	UF : 0, UT : 6,		CONFIG : 'N U T, 0, 0, 0',
	X =  19.695  mm,	Y =   -632.408  mm,	Z =   -236.035  mm,
	W =  90.000 deg,	P =   0.000 deg,	R =   90.000 deg
};
P[1150]{
   GP1:
	UF : 0, UT : 6,		CONFIG : 'N U T, 0, 0, 0',
	X =  20.066  mm,	Y =   -632.890  mm,	Z =   -236.261  mm,
	W =  90.000 deg,	P =   0.000 deg,	R =   90.000 deg
};
P[1151]{
   GP1:
	UF : 0, UT : 6,		CONFIG : 'N U T, 0, 0, 0',
	X =  21.473  mm,	Y =   -635.520  mm,	Z =   -235.987  mm,
	W =  90.000 deg,	P =   0.000 deg,	R =   90.000 deg
};
P[1152]{
   GP1:
	UF : 0, UT : 6,		CONFIG : 'N U T, 0, 0, 0',
	X =  22.170  mm,	Y =   -636.842  mm,	Z =   -235.830  mm,
	W =  90.000 deg,	P =   0.000 deg,	R =   90.000 deg
};
P[1153]{
   GP1:
	UF : 0, UT : 6,		CONFIG : 'N U T, 0, 0, 0',
	X =  22.857  mm,	Y =   -637.882  mm,	Z =   -236.036  mm,
	W =  90.000 deg,	P =   0.000 deg,	R =   90.000 deg
};
P[1154]{
   GP1:
	UF : 0, UT : 6,		CONFIG : 'N U T, 0, 0, 0',
	X =  25.259  mm,	Y =   -642.193  mm,	Z =   -235.826  mm,
	W =  90.000 deg,	P =   0.000 deg,	R =   90.000 deg
};
P[1155]{
   GP1:
	UF : 0, UT : 6,		CONFIG : 'N U T, 0, 0, 0',
	X =  26.183  mm,	Y =   -643.553  mm,	Z =   -236.163  mm,
	W =  90.000 deg,	P =   0.000 deg,	R =   90.000 deg
};
P[1156]{
   GP1:
	UF : 0, UT : 6,		CONFIG : 'N U T, 0, 0, 0',
	X =  26.417  mm,	Y =   -644.215  mm,	Z =   -235.804  mm,
	W =  90.000 deg,	P =   0.000 deg,	R =   90.000 deg
};
P[1157]{
   GP1:
	UF : 0, UT : 6,		CONFIG : 'N U T, 0, 0, 0',
	X =  27.412  mm,	Y =   -645.826  mm,	Z =   -235.959  mm,
	W =  90.000 deg,	P =   0.000 deg,	R =   90.000 deg
};
P[1158]{
   GP1:
	UF : 0, UT : 6,		CONFIG : 'N U T, 0, 0, 0',
	X =  28.982  mm,	Y =   -648.431  mm,	Z =   -236.122  mm,
	W =  90.000 deg,	P =   0.000 deg,	R =   90.000 deg
};
P[1159]{
   GP1:
	UF : 0, UT : 6,		CONFIG : 'N U T, 0, 0, 0',
	X =  29.599  mm,	Y =   -649.401  mm,	Z =   -236.259  mm,
	W =  90.000 deg,	P =   0.000 deg,	R =   90.000 deg
};
P[1160]{
   GP1:
	UF : 0, UT : 6,		CONFIG : 'N U T, 0, 0, 0',
	X =  30.088  mm,	Y =   -650.463  mm,	Z =   -235.958  mm,
	W =  90.000 deg,	P =   0.000 deg,	R =   90.000 deg
};
P[1161]{
   GP1:
	UF : 0, UT : 6,		CONFIG : 'N U T, 0, 0, 0',
	X =  30.788  mm,	Y =   -651.725  mm,	Z =   -235.889  mm,
	W =  90.000 deg,	P =   0.000 deg,	R =   90.000 deg
};
P[1162]{
   GP1:
	UF : 0, UT : 6,		CONFIG : 'N U T, 0, 0, 0',
	X =  31.326  mm,	Y =   -652.437  mm,	Z =   -236.196  mm,
	W =  90.000 deg,	P =   0.000 deg,	R =   90.000 deg
};
P[1163]{
   GP1:
	UF : 0, UT : 6,		CONFIG : 'N U T, 0, 0, 0',
	X =  33.837  mm,	Y =   -656.822  mm,	Z =   -236.144  mm,
	W =  90.000 deg,	P =   0.000 deg,	R =   90.000 deg
};
P[1164]{
   GP1:
	UF : 0, UT : 6,		CONFIG : 'N U T, 0, 0, 0',
	X =  34.171  mm,	Y =   -657.333  mm,	Z =   -236.240  mm,
	W =  90.000 deg,	P =   0.000 deg,	R =   90.000 deg
};
P[1165]{
   GP1:
	UF : 0, UT : 6,		CONFIG : 'N U T, 0, 0, 0',
	X =  35.312  mm,	Y =   -659.302  mm,	Z =   -236.251  mm,
	W =  90.000 deg,	P =   0.000 deg,	R =   90.000 deg
};
P[1166]{
   GP1:
	UF : 0, UT : 6,		CONFIG : 'N U T, 0, 0, 0',
	X =  36.261  mm,	Y =   -661.175  mm,	Z =   -235.927  mm,
	W =  90.000 deg,	P =   0.000 deg,	R =   90.000 deg
};
P[1167]{
   GP1:
	UF : 0, UT : 6,		CONFIG : 'N U T, 0, 0, 0',
	X =  36.673  mm,	Y =   -661.862  mm,	Z =   -235.965  mm,
	W =  90.000 deg,	P =   0.000 deg,	R =   90.000 deg
};
P[1168]{
   GP1:
	UF : 0, UT : 6,		CONFIG : 'N U T, 0, 0, 0',
	X =  37.452  mm,	Y =   -663.236  mm,	Z =   -235.932  mm,
	W =  90.000 deg,	P =   0.000 deg,	R =   90.000 deg
};
P[1169]{
   GP1:
	UF : 0, UT : 6,		CONFIG : 'N U T, 0, 0, 0',
	X =  38.851  mm,	Y =   -665.730  mm,	Z =   -235.831  mm,
	W =  90.000 deg,	P =   0.000 deg,	R =   90.000 deg
};
P[1170]{
   GP1:
	UF : 0, UT : 6,		CONFIG : 'N U T, 0, 0, 0',
	X =  39.817  mm,	Y =   -667.148  mm,	Z =   -236.188  mm,
	W =  90.000 deg,	P =   0.000 deg,	R =   90.000 deg
};
P[1171]{
   GP1:
	UF : 0, UT : 6,		CONFIG : 'N U T, 0, 0, 0',
	X =  41.225  mm,	Y =   -669.627  mm,	Z =   -236.131  mm,
	W =  90.000 deg,	P =   0.000 deg,	R =   90.000 deg
};
P[1172]{
   GP1:
	UF : 0, UT : 6,		CONFIG : 'N U T, 0, 0, 0',
	X =  41.505  mm,	Y =   -670.293  mm,	Z =   -235.877  mm,
	W =  90.000 deg,	P =   0.000 deg,	R =   90.000 deg
};
P[1173]{
   GP1:
	UF : 0, UT : 6,		CONFIG : 'N U T, 0, 0, 0',
	X =  42.466  mm,	Y =   -671.763  mm,	Z =   -236.150  mm,
	W =  90.000 deg,	P =   0.000 deg,	R =   90.000 deg
};
P[1174]{
   GP1:
	UF : 0, UT : 6,		CONFIG : 'N U T, 0, 0, 0',
	X =  44.206  mm,	Y =   -675.025  mm,	Z =   -235.802  mm,
	W =  90.000 deg,	P =   0.000 deg,	R =   90.000 deg
};
P[1175]{
   GP1:
	UF : 0, UT : 6,		CONFIG : 'N U T, 0, 0, 0',
	X =  45.308  mm,	Y =   -676.876  mm,	Z =   -235.884  mm,
	W =  90.000 deg,	P =   0.000 deg,	R =   90.000 deg
};
P[1176]{
   GP1:
	UF : 0, UT : 6,		CONFIG : 'N U T, 0, 0, 0',
	X =  48.322  mm,	Y =   -681.161  mm,	Z =   -236.219  mm,
	W =  90.000 deg,	P =   0.000 deg,	R =   90.000 deg
};
P[1177]{
   GP1:
	UF : 0, UT : 6,		CONFIG : 'N U T, 0, 0, 0',
	X =  48.985  mm,	Y =   -682.066  mm,	Z =   -235.767  mm,
	W =  90.000 deg,	P =   0.000 deg,	R =   90.000 deg
};
P[1178]{
   GP1:
	UF : 0, UT : 6,		CONFIG : 'N U T, 0, 0, 0',
	X =  50.468  mm,	Y =   -683.145  mm,	Z =   -236.020  mm,
	W =  90.000 deg,	P =   0.000 deg,	R =   90.000 deg
};
P[1179]{
   GP1:
	UF : 0, UT : 6,		CONFIG : 'N U T, 0, 0, 0',
	X =  52.789  mm,	Y =   -684.503  mm,	Z =   -235.854  mm,
	W =  90.000 deg,	P =   0.000 deg,	R =   90.000 deg
};
P[1180]{
   GP1:
	UF : 0, UT : 6,		CONFIG : 'N U T, 0, 0, 0',
	X =  57.085  mm,	Y =   -685.239  mm,	Z =   -236.177  mm,
	W =  90.000 deg,	P =   0.000 deg,	R =   90.000 deg
};
P[1181]{
   GP1:
	UF : 0, UT : 6,		CONFIG : 'N U T, 0, 0, 0',
	X =  59.311  mm,	Y =   -685.278  mm,	Z =   -235.865  mm,
	W =  90.000 deg,	P =   0.000 deg,	R =   90.000 deg
};
P[1182]{
   GP1:
	UF : 0, UT : 6,		CONFIG : 'N U T, 0, 0, 0',
	X =  60.413  mm,	Y =   -684.908  mm,	Z =   -236.185  mm,
	W =  90.000 deg,	P =   0.000 deg,	R =   90.000 deg
};
P[1183]{
   GP1:
	UF : 0, UT : 6,		CONFIG : 'N U T, 0, 0, 0',
	X =  61.691  mm,	Y =   -684.746  mm,	Z =   -235.808  mm,
	W =  90.000 deg,	P =   0.000 deg,	R =   90.000 deg
};
P[1184]{
   GP1:
	UF : 0, UT : 6,		CONFIG : 'N U T, 0, 0, 0',
	X =  62.508  mm,	Y =   -684.214  mm,	Z =   -236.201  mm,
	W =  90.000 deg,	P =   0.000 deg,	R =   90.000 deg
};
P[1185]{
   GP1:
	UF : 0, UT : 6,		CONFIG : 'N U T, 0, 0, 0',
	X =  63.457  mm,	Y =   -683.779  mm,	Z =   -236.224  mm,
	W =  90.000 deg,	P =   0.000 deg,	R =   90.000 deg
};
P[1186]{
   GP1:
	UF : 0, UT : 6,		CONFIG : 'N U T, 0, 0, 0',
	X =  64.865  mm,	Y =   -683.047  mm,	Z =   -236.231  mm,
	W =  90.000 deg,	P =   0.000 deg,	R =   90.000 deg
};
P[1187]{
   GP1:
	UF : 0, UT : 6,		CONFIG : 'N U T, 0, 0, 0',
	X =  66.260  mm,	Y =   -682.344  mm,	Z =   -235.984  mm,
	W =  90.000 deg,	P =   0.000 deg,	R =   90.000 deg
};
P[1188]{
   GP1:
	UF : 0, UT : 6,		CONFIG : 'N U T, 0, 0, 0',
	X =  68.438  mm,	Y =   -681.119  mm,	Z =   -235.906  mm,
	W =  90.000 deg,	P =   0.000 deg,	R =   90.000 deg
};
P[1189]{
   GP1:
	UF : 0, UT : 6,		CONFIG : 'N U T, 0, 0, 0',
	X =  71.774  mm,	Y =   -679.075  mm,	Z =   -236.192  mm,
	W =  90.000 deg,	P =   0.000 deg,	R =   90.000 deg
};
P[1190]{
   GP1:
	UF : 0, UT : 6,		CONFIG : 'N U T, 0, 0, 0',
	X =  72.829  mm,	Y =   -678.491  mm,	Z =   -236.131  mm,
	W =  90.000 deg,	P =   0.000 deg,	R =   90.000 deg
};
P[1191]{
   GP1:
	UF : 0, UT : 6,		CONFIG : 'N U T, 0, 0, 0',
	X =  75.444  mm,	Y =   -677.073  mm,	Z =   -235.905  mm,
	W =  90.000 deg,	P =   0.000 deg,	R =   90.000 deg
};
P[1192]{
   GP1:
	UF : 0, UT : 6,		CONFIG : 'N U T, 0, 0, 0',
	X =  76.617  mm,	Y =   -676.318  mm,	Z =   -236.096  mm,
	W =  90.000 deg,	P =   0.000 deg,	R =   90.000 deg
};
P[1193]{
   GP1:
	UF : 0, UT : 6,		CONFIG : 'N U T, 0, 0, 0',
	X =  82.666  mm,	Y =   -672.836  mm,	Z =   -236.069  mm,
	W =  90.000 deg,	P =   0.000 deg,	R =   90.000 deg
};
P[1194]{
   GP1:
	UF : 0, UT : 6,		CONFIG : 'N U T, 0, 0, 0',
	X =  83.579  mm,	Y =   -672.339  mm,	Z =   -235.997  mm,
	W =  90.000 deg,	P =   0.000 deg,	R =   90.000 deg
};
P[1195]{
   GP1:
	UF : 0, UT : 6,		CONFIG : 'N U T, 0, 0, 0',
	X =  84.352  mm,	Y =   -671.819  mm,	Z =   -236.176  mm,
	W =  90.000 deg,	P =   0.000 deg,	R =   90.000 deg
};
P[1196]{
   GP1:
	UF : 0, UT : 6,		CONFIG : 'N U T, 0, 0, 0',
	X =  86.806  mm,	Y =   -670.389  mm,	Z =   -236.207  mm,
	W =  90.000 deg,	P =   0.000 deg,	R =   90.000 deg
};
P[1197]{
   GP1:
	UF : 0, UT : 6,		CONFIG : 'N U T, 0, 0, 0',
	X =  87.702  mm,	Y =   -669.881  mm,	Z =   -236.187  mm,
	W =  90.000 deg,	P =   0.000 deg,	R =   90.000 deg
};
P[1198]{
   GP1:
	UF : 0, UT : 6,		CONFIG : 'N U T, 0, 0, 0',
	X =  91.684  mm,	Y =   -667.560  mm,	Z =   -236.236  mm,
	W =  90.000 deg,	P =   0.000 deg,	R =   90.000 deg
};
P[1199]{
   GP1:
	UF : 0, UT : 6,		CONFIG : 'N U T, 0, 0, 0',
	X =  92.871  mm,	Y =   -666.995  mm,	Z =   -235.945  mm,
	W =  90.000 deg,	P =   0.000 deg,	R =   90.000 deg
};
P[1200]{
   GP1:
	UF : 0, UT : 6,		CONFIG : 'N U T, 0, 0, 0',
	X =  93.918  mm,	Y =   -666.295  mm,	Z =   -236.177  mm,
	W =  90.000 deg,	P =   0.000 deg,	R =   90.000 deg
};
P[1201]{
   GP1:
	UF : 0, UT : 6,		CONFIG : 'N U T, 0, 0, 0',
	X =  96.550  mm,	Y =   -664.748  mm,	Z =   -236.242  mm,
	W =  90.000 deg,	P =   0.000 deg,	R =   90.000 deg
};
P[1202]{
   GP1:
	UF : 0, UT : 6,		CONFIG : 'N U T, 0, 0, 0',
	X =  98.885  mm,	Y =   -663.545  mm,	Z =   -235.890  mm,
	W =  90.000 deg,	P =   0.000 deg,	R =   90.000 deg
};
P[1203]{
   GP1:
	UF : 0, UT : 6,		CONFIG : 'N U T, 0, 0, 0',
	X =  101.949  mm,	Y =   -661.786  mm,	Z =   -235.866  mm,
	W =  90.000 deg,	P =   0.000 deg,	R =   90.000 deg
};
P[1204]{
   GP1:
	UF : 0, UT : 6,		CONFIG : 'N U T, 0, 0, 0',
	X =  105.049  mm,	Y =   -659.837  mm,	Z =   -236.252  mm,
	W =  90.000 deg,	P =   0.000 deg,	R =   90.000 deg
};
P[1205]{
   GP1:
	UF : 0, UT : 6,		CONFIG : 'N U T, 0, 0, 0',
	X =  107.967  mm,	Y =   -658.192  mm,	Z =   -236.155  mm,
	W =  90.000 deg,	P =   0.000 deg,	R =   90.000 deg
};
P[1206]{
   GP1:
	UF : 0, UT : 6,		CONFIG : 'N U T, 0, 0, 0',
	X =  109.064  mm,	Y =   -657.606  mm,	Z =   -236.039  mm,
	W =  90.000 deg,	P =   0.000 deg,	R =   90.000 deg
};
P[1207]{
   GP1:
	UF : 0, UT : 6,		CONFIG : 'N U T, 0, 0, 0',
	X =  110.455  mm,	Y =   -656.731  mm,	Z =   -236.216  mm,
	W =  90.000 deg,	P =   0.000 deg,	R =   90.000 deg
};
P[1208]{
   GP1:
	UF : 0, UT : 6,		CONFIG : 'N U T, 0, 0, 0',
	X =  113.229  mm,	Y =   -655.189  mm,	Z =   -236.069  mm,
	W =  90.000 deg,	P =   0.000 deg,	R =   90.000 deg
};
P[1209]{
   GP1:
	UF : 0, UT : 6,		CONFIG : 'N U T, 0, 0, 0',
	X =  115.613  mm,	Y =   -653.845  mm,	Z =   -235.990  mm,
	W =  90.000 deg,	P =   0.000 deg,	R =   90.000 deg
};
P[1210]{
   GP1:
	UF : 0, UT : 6,		CONFIG : 'N U T, 0, 0, 0',
	X =  120.896  mm,	Y =   -650.754  mm,	Z =   -236.090  mm,
	W =  90.000 deg,	P =   0.000 deg,	R =   90.000 deg
};
P[1211]{
   GP1:
	UF : 0, UT : 6,		CONFIG : 'N U T, 0, 0, 0',
	X =  122.286  mm,	Y =   -649.951  mm,	Z =   -236.092  mm,
	W =  90.000 deg,	P =   0.000 deg,	R =   90.000 deg
};
P[1212]{
   GP1:
	UF : 0, UT : 6,		CONFIG : 'N U T, 0, 0, 0',
	X =  128.537  mm,	Y =   -646.275  mm,	Z =   -236.252  mm,
	W =  90.000 deg,	P =   0.000 deg,	R =   90.000 deg
};
P[1213]{
   GP1:
	UF : 0, UT : 6,		CONFIG : 'N U T, 0, 0, 0',
	X =  129.609  mm,	Y =   -645.663  mm,	Z =   -236.237  mm,
	W =  90.000 deg,	P =   0.000 deg,	R =   90.000 deg
};
P[1214]{
   GP1:
	UF : 0, UT : 6,		CONFIG : 'N U T, 0, 0, 0',
	X =  130.636  mm,	Y =   -645.107  mm,	Z =   -236.148  mm,
	W =  90.000 deg,	P =   0.000 deg,	R =   90.000 deg
};
P[1215]{
   GP1:
	UF : 0, UT : 6,		CONFIG : 'N U T, 0, 0, 0',
	X =  131.238  mm,	Y =   -644.736  mm,	Z =   -236.204  mm,
	W =  90.000 deg,	P =   0.000 deg,	R =   90.000 deg
};
P[1216]{
   GP1:
	UF : 0, UT : 6,		CONFIG : 'N U T, 0, 0, 0',
	X =  135.205  mm,	Y =   -642.495  mm,	Z =   -236.084  mm,
	W =  90.000 deg,	P =   0.000 deg,	R =   90.000 deg
};
P[1217]{
   GP1:
	UF : 0, UT : 6,		CONFIG : 'N U T, 0, 0, 0',
	X =  138.112  mm,	Y =   -640.947  mm,	Z =   -235.765  mm,
	W =  90.000 deg,	P =   0.000 deg,	R =   90.000 deg
};
P[1218]{
   GP1:
	UF : 0, UT : 6,		CONFIG : 'N U T, 0, 0, 0',
	X =  139.022  mm,	Y =   -640.231  mm,	Z =   -236.231  mm,
	W =  90.000 deg,	P =   0.000 deg,	R =   90.000 deg
};
P[1219]{
   GP1:
	UF : 0, UT : 6,		CONFIG : 'N U T, 0, 0, 0',
	X =  140.803  mm,	Y =   -639.313  mm,	Z =   -235.959  mm,
	W =  90.000 deg,	P =   0.000 deg,	R =   90.000 deg
};
P[1220]{
   GP1:
	UF : 0, UT : 6,		CONFIG : 'N U T, 0, 0, 0',
	X =  141.464  mm,	Y =   -638.891  mm,	Z =   -236.060  mm,
	W =  90.000 deg,	P =   0.000 deg,	R =   90.000 deg
};
P[1221]{
   GP1:
	UF : 0, UT : 6,		CONFIG : 'N U T, 0, 0, 0',
	X =  144.134  mm,	Y =   -637.401  mm,	Z =   -235.935  mm,
	W =  90.000 deg,	P =   0.000 deg,	R =   90.000 deg
};
P[1222]{
   GP1:
	UF : 0, UT : 6,		CONFIG : 'N U T, 0, 0, 0',
	X =  145.036  mm,	Y =   -636.806  mm,	Z =   -236.112  mm,
	W =  90.000 deg,	P =   0.000 deg,	R =   90.000 deg
};
P[1223]{
   GP1:
	UF : 0, UT : 6,		CONFIG : 'N U T, 0, 0, 0',
	X =  145.813  mm,	Y =   -636.296  mm,	Z =   -236.263  mm,
	W =  90.000 deg,	P =   0.000 deg,	R =   90.000 deg
};
P[1224]{
   GP1:
	UF : 0, UT : 6,		CONFIG : 'N U T, 0, 0, 0',
	X =  147.022  mm,	Y =   -635.665  mm,	Z =   -236.101  mm,
	W =  90.000 deg,	P =   0.000 deg,	R =   90.000 deg
};
P[1225]{
   GP1:
	UF : 0, UT : 6,		CONFIG : 'N U T, 0, 0, 0',
	X =  148.140  mm,	Y =   -635.017  mm,	Z =   -236.107  mm,
	W =  90.000 deg,	P =   0.000 deg,	R =   90.000 deg
};
P[1226]{
   GP1:
	UF : 0, UT : 6,		CONFIG : 'N U T, 0, 0, 0',
	X =  149.297  mm,	Y =   -634.466  mm,	Z =   -235.820  mm,
	W =  90.000 deg,	P =   0.000 deg,	R =   90.000 deg
};
P[1227]{
   GP1:
	UF : 0, UT : 6,		CONFIG : 'N U T, 0, 0, 0',
	X =  152.287  mm,	Y =   -632.743  mm,	Z =   -235.814  mm,
	W =  90.000 deg,	P =   0.000 deg,	R =   90.000 deg
};
P[1228]{
   GP1:
	UF : 0, UT : 6,		CONFIG : 'N U T, 0, 0, 0',
	X =  153.491  mm,	Y =   -631.907  mm,	Z =   -236.155  mm,
	W =  90.000 deg,	P =   0.000 deg,	R =   90.000 deg
};
P[1229]{
   GP1:
	UF : 0, UT : 6,		CONFIG : 'N U T, 0, 0, 0',
	X =  154.682  mm,	Y =   -631.302  mm,	Z =   -235.956  mm,
	W =  90.000 deg,	P =   0.000 deg,	R =   90.000 deg
};
P[1230]{
   GP1:
	UF : 0, UT : 6,		CONFIG : 'N U T, 0, 0, 0',
	X =  155.626  mm,	Y =   -630.706  mm,	Z =   -236.079  mm,
	W =  90.000 deg,	P =   0.000 deg,	R =   90.000 deg
};
P[1231]{
   GP1:
	UF : 0, UT : 6,		CONFIG : 'N U T, 0, 0, 0',
	X =  157.770  mm,	Y =   -629.514  mm,	Z =   -235.969  mm,
	W =  90.000 deg,	P =   0.000 deg,	R =   90.000 deg
};
P[1232]{
   GP1:
	UF : 0, UT : 6,		CONFIG : 'N U T, 0, 0, 0',
	X =  160.528  mm,	Y =   -627.937  mm,	Z =   -235.928  mm,
	W =  90.000 deg,	P =   0.000 deg,	R =   90.000 deg
};
P[1233]{
   GP1:
	UF : 0, UT : 6,		CONFIG : 'N U T, 0, 0, 0',
	X =  161.238  mm,	Y =   -627.424  mm,	Z =   -236.177  mm,
	W =  90.000 deg,	P =   0.000 deg,	R =   90.000 deg
};
P[1234]{
   GP1:
	UF : 0, UT : 6,		CONFIG : 'N U T, 0, 0, 0',
	X =  162.012  mm,	Y =   -627.052  mm,	Z =   -235.999  mm,
	W =  90.000 deg,	P =   0.000 deg,	R =   90.000 deg
};
P[1235]{
   GP1:
	UF : 0, UT : 6,		CONFIG : 'N U T, 0, 0, 0',
	X =  166.933  mm,	Y =   -624.102  mm,	Z =   -236.262  mm,
	W =  90.000 deg,	P =   0.000 deg,	R =   90.000 deg
};
P[1236]{
   GP1:
	UF : 0, UT : 6,		CONFIG : 'N U T, 0, 0, 0',
	X =  167.569  mm,	Y =   -623.749  mm,	Z =   -236.228  mm,
	W =  90.000 deg,	P =   0.000 deg,	R =   90.000 deg
};
P[1237]{
   GP1:
	UF : 0, UT : 6,		CONFIG : 'N U T, 0, 0, 0',
	X =  170.488  mm,	Y =   -622.121  mm,	Z =   -236.089  mm,
	W =  90.000 deg,	P =   0.000 deg,	R =   90.000 deg
};
P[1238]{
   GP1:
	UF : 0, UT : 6,		CONFIG : 'N U T, 0, 0, 0',
	X =  171.115  mm,	Y =   -621.725  mm,	Z =   -236.171  mm,
	W =  90.000 deg,	P =   0.000 deg,	R =   90.000 deg
};
P[1239]{
   GP1:
	UF : 0, UT : 6,		CONFIG : 'N U T, 0, 0, 0',
	X =  171.685  mm,	Y =   -621.363  mm,	Z =   -236.249  mm,
	W =  90.000 deg,	P =   0.000 deg,	R =   90.000 deg
};
P[1240]{
   GP1:
	UF : 0, UT : 6,		CONFIG : 'N U T, 0, 0, 0',
	X =  176.974  mm,	Y =   -618.470  mm,	Z =   -235.859  mm,
	W =  90.000 deg,	P =   0.000 deg,	R =   90.000 deg
};
P[1241]{
   GP1:
	UF : 0, UT : 6,		CONFIG : 'N U T, 0, 0, 0',
	X =  178.817  mm,	Y =   -617.389  mm,	Z =   -235.902  mm,
	W =  90.000 deg,	P =   0.000 deg,	R =   90.000 deg
};
P[1242]{
   GP1:
	UF : 0, UT : 6,		CONFIG : 'N U T, 0, 0, 0',
	X =  182.698  mm,	Y =   -615.137  mm,	Z =   -235.927  mm,
	W =  90.000 deg,	P =   0.000 deg,	R =   90.000 deg
};
P[1243]{
   GP1:
	UF : 0, UT : 6,		CONFIG : 'N U T, 0, 0, 0',
	X =  187.118  mm,	Y =   -612.467  mm,	Z =   -236.214  mm,
	W =  90.000 deg,	P =   0.000 deg,	R =   90.000 deg
};
P[1244]{
   GP1:
	UF : 0, UT : 6,		CONFIG : 'N U T, 0, 0, 0',
	X =  190.558  mm,	Y =   -610.460  mm,	Z =   -236.263  mm,
	W =  90.000 deg,	P =   0.000 deg,	R =   90.000 deg
};
P[1245]{
   GP1:
	UF : 0, UT : 6,		CONFIG : 'N U T, 0, 0, 0',
	X =  194.089  mm,	Y =   -608.591  mm,	Z =   -235.851  mm,
	W =  90.000 deg,	P =   0.000 deg,	R =   90.000 deg
};
P[1246]{
   GP1:
	UF : 0, UT : 6,		CONFIG : 'N U T, 0, 0, 0',
	X =  195.296  mm,	Y =   -607.726  mm,	Z =   -236.259  mm,
	W =  90.000 deg,	P =   0.000 deg,	R =   90.000 deg
};
P[1247]{
   GP1:
	UF : 0, UT : 6,		CONFIG : 'N U T, 0, 0, 0',
	X =  197.817  mm,	Y =   -606.299  mm,	Z =   -236.192  mm,
	W =  90.000 deg,	P =   0.000 deg,	R =   90.000 deg
};
P[1248]{
   GP1:
	UF : 0, UT : 6,		CONFIG : 'N U T, 0, 0, 0',
	X =  201.527  mm,	Y =   -604.217  mm,	Z =   -236.045  mm,
	W =  90.000 deg,	P =   0.000 deg,	R =   90.000 deg
};
P[1249]{
   GP1:
	UF : 0, UT : 6,		CONFIG : 'N U T, 0, 0, 0',
	X =  203.422  mm,	Y =   -603.063  mm,	Z =   -236.190  mm,
	W =  90.000 deg,	P =   0.000 deg,	R =   90.000 deg
};
P[1250]{
   GP1:
	UF : 0, UT : 6,		CONFIG : 'N U T, 0, 0, 0',
	X =  205.460  mm,	Y =   -602.039  mm,	Z =   -235.818  mm,
	W =  90.000 deg,	P =   0.000 deg,	R =   90.000 deg
};
P[1251]{
   GP1:
	UF : 0, UT : 6,		CONFIG : 'N U T, 0, 0, 0',
	X =  207.396  mm,	Y =   -600.770  mm,	Z =   -236.186  mm,
	W =  90.000 deg,	P =   0.000 deg,	R =   90.000 deg
};
P[1252]{
   GP1:
	UF : 0, UT : 6,		CONFIG : 'N U T, 0, 0, 0',
	X =  208.921  mm,	Y =   -599.898  mm,	Z =   -236.166  mm,
	W =  90.000 deg,	P =   0.000 deg,	R =   90.000 deg
};
P[1253]{
   GP1:
	UF : 0, UT : 6,		CONFIG : 'N U T, 0, 0, 0',
	X =  214.058  mm,	Y =   -596.930  mm,	Z =   -236.170  mm,
	W =  90.000 deg,	P =   0.000 deg,	R =   90.000 deg
};
P[1254]{
   GP1:
	UF : 0, UT : 6,		CONFIG : 'N U T, 0, 0, 0',
	X =  215.411  mm,	Y =   -596.265  mm,	Z =   -235.888  mm,
	W =  90.000 deg,	P =   0.000 deg,	R =   90.000 deg
};
P[1255]{
   GP1:
	UF : 0, UT : 6,		CONFIG : 'N U T, 0, 0, 0',
	X =  216.083  mm,	Y =   -595.781  mm,	Z =   -236.121  mm,
	W =  90.000 deg,	P =   0.000 deg,	R =   90.000 deg
};
P[1256]{
   GP1:
	UF : 0, UT : 6,		CONFIG : 'N U T, 0, 0, 0',
	X =  217.510  mm,	Y =   -595.040  mm,	Z =   -235.921  mm,
	W =  90.000 deg,	P =   0.000 deg,	R =   90.000 deg
};
P[1257]{
   GP1:
	UF : 0, UT : 6,		CONFIG : 'N U T, 0, 0, 0',
	X =  218.922  mm,	Y =   -594.257  mm,	Z =   -235.842  mm,
	W =  90.000 deg,	P =   0.000 deg,	R =   90.000 deg
};
P[1258]{
   GP1:
	UF : 0, UT : 6,		CONFIG : 'N U T, 0, 0, 0',
	X =  220.028  mm,	Y =   -593.525  mm,	Z =   -236.068  mm,
	W =  90.000 deg,	P =   0.000 deg,	R =   90.000 deg
};
P[1259]{
   GP1:
	UF : 0, UT : 6,		CONFIG : 'N U T, 0, 0, 0',
	X =  220.868  mm,	Y =   -592.976  mm,	Z =   -236.224  mm,
	W =  90.000 deg,	P =   0.000 deg,	R =   90.000 deg
};
P[1260]{
   GP1:
	UF : 0, UT : 6,		CONFIG : 'N U T, 0, 0, 0',
	X =  221.717  mm,	Y =   -592.602  mm,	Z =   -235.941  mm,
	W =  90.000 deg,	P =   0.000 deg,	R =   90.000 deg
};
P[1261]{
   GP1:
	UF : 0, UT : 6,		CONFIG : 'N U T, 0, 0, 0',
	X =  227.339  mm,	Y =   -589.409  mm,	Z =   -235.814  mm,
	W =  90.000 deg,	P =   0.000 deg,	R =   90.000 deg
};
P[1262]{
   GP1:
	UF : 0, UT : 6,		CONFIG : 'N U T, 0, 0, 0',
	X =  227.893  mm,	Y =   -588.916  mm,	Z =   -236.232  mm,
	W =  90.000 deg,	P =   0.000 deg,	R =   90.000 deg
};
P[1263]{
   GP1:
	UF : 0, UT : 6,		CONFIG : 'N U T, 0, 0, 0',
	X =  229.324  mm,	Y =   -588.095  mm,	Z =   -236.219  mm,
	W =  90.000 deg,	P =   0.000 deg,	R =   90.000 deg
};
P[1264]{
   GP1:
	UF : 0, UT : 6,		CONFIG : 'N U T, 0, 0, 0',
	X =  230.255  mm,	Y =   -587.636  mm,	Z =   -236.030  mm,
	W =  90.000 deg,	P =   0.000 deg,	R =   90.000 deg
};
P[1265]{
   GP1:
	UF : 0, UT : 6,		CONFIG : 'N U T, 0, 0, 0',
	X =  231.063  mm,	Y =   -587.085  mm,	Z =   -236.234  mm,
	W =  90.000 deg,	P =   0.000 deg,	R =   90.000 deg
};
P[1266]{
   GP1:
	UF : 0, UT : 6,		CONFIG : 'N U T, 0, 0, 0',
	X =  232.274  mm,	Y =   -586.571  mm,	Z =   -235.786  mm,
	W =  90.000 deg,	P =   0.000 deg,	R =   90.000 deg
};
P[1267]{
   GP1:
	UF : 0, UT : 6,		CONFIG : 'N U T, 0, 0, 0',
	X =  234.541  mm,	Y =   -585.154  mm,	Z =   -236.047  mm,
	W =  90.000 deg,	P =   0.000 deg,	R =   90.000 deg
};
P[1268]{
   GP1:
	UF : 0, UT : 6,		CONFIG : 'N U T, 0, 0, 0',
	X =  235.154  mm,	Y =   -584.834  mm,	Z =   -235.966  mm,
	W =  90.000 deg,	P =   0.000 deg,	R =   90.000 deg
};
P[1269]{
   GP1:
	UF : 0, UT : 6,		CONFIG : 'N U T, 0, 0, 0',
	X =  238.918  mm,	Y =   -582.572  mm,	Z =   -236.180  mm,
	W =  90.000 deg,	P =   0.000 deg,	R =   90.000 deg
};
P[1270]{
   GP1:
	UF : 0, UT : 6,		CONFIG : 'N U T, 0, 0, 0',
	X =  240.565  mm,	Y =   -581.599  mm,	Z =   -236.235  mm,
	W =  90.000 deg,	P =   0.000 deg,	R =   90.000 deg
};
P[1271]{
   GP1:
	UF : 0, UT : 6,		CONFIG : 'N U T, 0, 0, 0',
	X =  243.237  mm,	Y =   -580.142  mm,	Z =   -236.025  mm,
	W =  90.000 deg,	P =   0.000 deg,	R =   90.000 deg
};
P[1272]{
   GP1:
	UF : 0, UT : 6,		CONFIG : 'N U T, 0, 0, 0',
	X =  243.899  mm,	Y =   -579.691  mm,	Z =   -236.193  mm,
	W =  90.000 deg,	P =   0.000 deg,	R =   90.000 deg
};
P[1273]{
   GP1:
	UF : 0, UT : 6,		CONFIG : 'N U T, 0, 0, 0',
	X =  246.134  mm,	Y =   -578.564  mm,	Z =   -235.796  mm,
	W =  90.000 deg,	P =   0.000 deg,	R =   90.000 deg
};
P[1274]{
   GP1:
	UF : 0, UT : 6,		CONFIG : 'N U T, 0, 0, 0',
	X =  246.789  mm,	Y =   -578.068  mm,	Z =   -236.081  mm,
	W =  90.000 deg,	P =   0.000 deg,	R =   90.000 deg
};
P[1275]{
   GP1:
	UF : 0, UT : 6,		CONFIG : 'N U T, 0, 0, 0',
	X =  248.147  mm,	Y =   -577.360  mm,	Z =   -235.895  mm,
	W =  90.000 deg,	P =   0.000 deg,	R =   90.000 deg
};
P[1276]{
   GP1:
	UF : 0, UT : 6,		CONFIG : 'N U T, 0, 0, 0',
	X =  250.469  mm,	Y =   -575.911  mm,	Z =   -236.160  mm,
	W =  90.000 deg,	P =   0.000 deg,	R =   90.000 deg
};
P[1277]{
   GP1:
	UF : 0, UT : 6,		CONFIG : 'N U T, 0, 0, 0',
	X =  250.972  mm,	Y =   -575.776  mm,	Z =   -235.783  mm,
	W =  90.000 deg,	P =   0.000 deg,	R =   90.000 deg
};
P[1278]{
   GP1:
	UF : 0, UT : 6,		CONFIG : 'N U T, 0, 0, 0',
	X =  251.820  mm,	Y =   -575.114  mm,	Z =   -236.201  mm,
	W =  90.000 deg,	P =   0.000 deg,	R =   90.000 deg
};
P[1279]{
   GP1:
	UF : 0, UT : 6,		CONFIG : 'N U T, 0, 0, 0',
	X =  253.992  mm,	Y =   -573.920  mm,	Z =   -236.056  mm,
	W =  90.000 deg,	P =   0.000 deg,	R =   90.000 deg
};
P[1280]{
   GP1:
	UF : 0, UT : 6,		CONFIG : 'N U T, 0, 0, 0',
	X =  255.262  mm,	Y =   -573.131  mm,	Z =   -236.189  mm,
	W =  90.000 deg,	P =   0.000 deg,	R =   90.000 deg
};
P[1281]{
   GP1:
	UF : 0, UT : 6,		CONFIG : 'N U T, 0, 0, 0',
	X =  257.360  mm,	Y =   -571.996  mm,	Z =   -236.003  mm,
	W =  90.000 deg,	P =   0.000 deg,	R =   90.000 deg
};
P[1282]{
   GP1:
	UF : 0, UT : 6,		CONFIG : 'N U T, 0, 0, 0',
	X =  258.170  mm,	Y =   -571.487  mm,	Z =   -236.104  mm,
	W =  90.000 deg,	P =   0.000 deg,	R =   90.000 deg
};
P[1283]{
   GP1:
	UF : 0, UT : 6,		CONFIG : 'N U T, 0, 0, 0',
	X =  258.767  mm,	Y =   -571.157  mm,	Z =   -236.070  mm,
	W =  90.000 deg,	P =   0.000 deg,	R =   90.000 deg
};
P[1284]{
   GP1:
	UF : 0, UT : 6,		CONFIG : 'N U T, 0, 0, 0',
	X =  260.090  mm,	Y =   -570.509  mm,	Z =   -235.789  mm,
	W =  90.000 deg,	P =   0.000 deg,	R =   90.000 deg
};
P[1285]{
   GP1:
	UF : 0, UT : 6,		CONFIG : 'N U T, 0, 0, 0',
	X =  261.709  mm,	Y =   -569.511  mm,	Z =   -235.943  mm,
	W =  90.000 deg,	P =   0.000 deg,	R =   90.000 deg
};
P[1286]{
   GP1:
	UF : 0, UT : 6,		CONFIG : 'N U T, 0, 0, 0',
	X =  264.842  mm,	Y =   -567.577  mm,	Z =   -236.245  mm,
	W =  90.000 deg,	P =   0.000 deg,	R =   90.000 deg
};
P[1287]{
   GP1:
	UF : 0, UT : 6,		CONFIG : 'N U T, 0, 0, 0',
	X =  266.479  mm,	Y =   -566.667  mm,	Z =   -236.161  mm,
	W =  90.000 deg,	P =   0.000 deg,	R =   90.000 deg
};
P[1288]{
   GP1:
	UF : 0, UT : 6,		CONFIG : 'N U T, 0, 0, 0',
	X =  267.664  mm,	Y =   -565.952  mm,	Z =   -236.234  mm,
	W =  90.000 deg,	P =   0.000 deg,	R =   90.000 deg
};
P[1289]{
   GP1:
	UF : 0, UT : 6,		CONFIG : 'N U T, 0, 0, 0',
	X =  276.056  mm,	Y =   -561.178  mm,	Z =   -236.061  mm,
	W =  90.000 deg,	P =   0.000 deg,	R =   90.000 deg
};
P[1290]{
   GP1:
	UF : 0, UT : 6,		CONFIG : 'N U T, 0, 0, 0',
	X =  277.168  mm,	Y =   -560.537  mm,	Z =   -236.057  mm,
	W =  90.000 deg,	P =   0.000 deg,	R =   90.000 deg
};
P[1291]{
   GP1:
	UF : 0, UT : 6,		CONFIG : 'N U T, 0, 0, 0',
	X =  283.306  mm,	Y =   -556.934  mm,	Z =   -236.202  mm,
	W =  90.000 deg,	P =   0.000 deg,	R =   90.000 deg
};
P[1292]{
   GP1:
	UF : 0, UT : 6,		CONFIG : 'N U T, 0, 0, 0',
	X =  283.968  mm,	Y =   -556.545  mm,	Z =   -236.217  mm,
	W =  90.000 deg,	P =   0.000 deg,	R =   90.000 deg
};
P[1293]{
   GP1:
	UF : 0, UT : 6,		CONFIG : 'N U T, 0, 0, 0',
	X =  285.871  mm,	Y =   -555.459  mm,	Z =   -236.187  mm,
	W =  90.000 deg,	P =   0.000 deg,	R =   90.000 deg
};
P[1294]{
   GP1:
	UF : 0, UT : 6,		CONFIG : 'N U T, 0, 0, 0',
	X =  287.181  mm,	Y =   -554.798  mm,	Z =   -235.956  mm,
	W =  90.000 deg,	P =   0.000 deg,	R =   90.000 deg
};
P[1295]{
   GP1:
	UF : 0, UT : 6,		CONFIG : 'N U T, 0, 0, 0',
	X =  288.139  mm,	Y =   -554.117  mm,	Z =   -236.265  mm,
	W =  90.000 deg,	P =   0.000 deg,	R =   90.000 deg
};
P[1296]{
   GP1:
	UF : 0, UT : 6,		CONFIG : 'N U T, 0, 0, 0',
	X =  289.724  mm,	Y =   -553.246  mm,	Z =   -236.158  mm,
	W =  90.000 deg,	P =   0.000 deg,	R =   90.000 deg
};
P[1297]{
   GP1:
	UF : 0, UT : 6,		CONFIG : 'N U T, 0, 0, 0',
	X =  291.588  mm,	Y =   -552.148  mm,	Z =   -236.211  mm,
	W =  90.000 deg,	P =   0.000 deg,	R =   90.000 deg
};
P[1298]{
   GP1:
	UF : 0, UT : 6,		CONFIG : 'N U T, 0, 0, 0',
	X =  295.641  mm,	Y =   -549.911  mm,	Z =   -235.963  mm,
	W =  90.000 deg,	P =   0.000 deg,	R =   90.000 deg
};
P[1299]{
   GP1:
	UF : 0, UT : 6,		CONFIG : 'N U T, 0, 0, 0',
	X =  296.764  mm,	Y =   -549.341  mm,	Z =   -235.771  mm,
	W =  90.000 deg,	P =   0.000 deg,	R =   90.000 deg
};
P[1300]{
   GP1:
	UF : 0, UT : 6,		CONFIG : 'N U T, 0, 0, 0',
	X =  297.702  mm,	Y =   -548.664  mm,	Z =   -236.100  mm,
	W =  90.000 deg,	P =   0.000 deg,	R =   90.000 deg
};
P[1301]{
   GP1:
	UF : 0, UT : 6,		CONFIG : 'N U T, 0, 0, 0',
	X =  299.074  mm,	Y =   -547.841  mm,	Z =   -236.174  mm,
	W =  90.000 deg,	P =   0.000 deg,	R =   90.000 deg
};
P[1302]{
   GP1:
	UF : 0, UT : 6,		CONFIG : 'N U T, 0, 0, 0',
	X =  302.115  mm,	Y =   -546.189  mm,	Z =   -235.922  mm,
	W =  90.000 deg,	P =   0.000 deg,	R =   90.000 deg
};
P[1303]{
   GP1:
	UF : 0, UT : 6,		CONFIG : 'N U T, 0, 0, 0',
	X =  304.281  mm,	Y =   -544.967  mm,	Z =   -235.853  mm,
	W =  90.000 deg,	P =   0.000 deg,	R =   90.000 deg
};
P[1304]{
   GP1:
	UF : 0, UT : 6,		CONFIG : 'N U T, 0, 0, 0',
	X =  305.391  mm,	Y =   -544.285  mm,	Z =   -235.952  mm,
	W =  90.000 deg,	P =   0.000 deg,	R =   90.000 deg
};
P[1305]{
   GP1:
	UF : 0, UT : 6,		CONFIG : 'N U T, 0, 0, 0',
	X =  307.431  mm,	Y =   -543.087  mm,	Z =   -236.003  mm,
	W =  90.000 deg,	P =   0.000 deg,	R =   90.000 deg
};
P[1306]{
   GP1:
	UF : 0, UT : 6,		CONFIG : 'N U T, 0, 0, 0',
	X =  311.087  mm,	Y =   -540.904  mm,	Z =   -236.176  mm,
	W =  90.000 deg,	P =   0.000 deg,	R =   90.000 deg
};
P[1307]{
   GP1:
	UF : 0, UT : 6,		CONFIG : 'N U T, 0, 0, 0',
	X =  313.813  mm,	Y =   -539.340  mm,	Z =   -236.153  mm,
	W =  90.000 deg,	P =   0.000 deg,	R =   90.000 deg
};
P[1308]{
   GP1:
	UF : 0, UT : 6,		CONFIG : 'N U T, 0, 0, 0',
	X =  316.236  mm,	Y =   -537.898  mm,	Z =   -236.255  mm,
	W =  90.000 deg,	P =   0.000 deg,	R =   90.000 deg
};
P[1309]{
   GP1:
	UF : 0, UT : 6,		CONFIG : 'N U T, 0, 0, 0',
	X =  317.798  mm,	Y =   -536.997  mm,	Z =   -236.256  mm,
	W =  90.000 deg,	P =   0.000 deg,	R =   90.000 deg
};
P[1310]{
   GP1:
	UF : 0, UT : 6,		CONFIG : 'N U T, 0, 0, 0',
	X =  318.889  mm,	Y =   -536.446  mm,	Z =   -236.063  mm,
	W =  90.000 deg,	P =   0.000 deg,	R =   90.000 deg
};
P[1311]{
   GP1:
	UF : 0, UT : 6,		CONFIG : 'N U T, 0, 0, 0',
	X =  319.712  mm,	Y =   -535.896  mm,	Z =   -236.245  mm,
	W =  90.000 deg,	P =   0.000 deg,	R =   90.000 deg
};
P[1312]{
   GP1:
	UF : 0, UT : 6,		CONFIG : 'N U T, 0, 0, 0',
	X =  321.761  mm,	Y =   -534.847  mm,	Z =   -235.919  mm,
	W =  90.000 deg,	P =   0.000 deg,	R =   90.000 deg
};
P[1313]{
   GP1:
	UF : 0, UT : 6,		CONFIG : 'N U T, 0, 0, 0',
	X =  323.593  mm,	Y =   -533.676  mm,	Z =   -236.192  mm,
	W =  90.000 deg,	P =   0.000 deg,	R =   90.000 deg
};
P[1314]{
   GP1:
	UF : 0, UT : 6,		CONFIG : 'N U T, 0, 0, 0',
	X =  328.811  mm,	Y =   -530.729  mm,	Z =   -236.034  mm,
	W =  90.000 deg,	P =   0.000 deg,	R =   90.000 deg
};
P[1315]{
   GP1:
	UF : 0, UT : 6,		CONFIG : 'N U T, 0, 0, 0',
	X =  331.545  mm,	Y =   -529.062  mm,	Z =   -236.246  mm,
	W =  90.000 deg,	P =   0.000 deg,	R =   90.000 deg
};
P[1316]{
   GP1:
	UF : 0, UT : 6,		CONFIG : 'N U T, 0, 0, 0',
	X =  332.941  mm,	Y =   -528.255  mm,	Z =   -236.250  mm,
	W =  90.000 deg,	P =   0.000 deg,	R =   90.000 deg
};
P[1317]{
   GP1:
	UF : 0, UT : 6,		CONFIG : 'N U T, 0, 0, 0',
	X =  336.586  mm,	Y =   -526.149  mm,	Z =   -236.254  mm,
	W =  90.000 deg,	P =   0.000 deg,	R =   90.000 deg
};
P[1318]{
   GP1:
	UF : 0, UT : 6,		CONFIG : 'N U T, 0, 0, 0',
	X =  339.977  mm,	Y =   -524.251  mm,	Z =   -236.109  mm,
	W =  90.000 deg,	P =   0.000 deg,	R =   90.000 deg
};
P[1319]{
   GP1:
	UF : 0, UT : 6,		CONFIG : 'N U T, 0, 0, 0',
	X =  341.795  mm,	Y =   -523.168  mm,	Z =   -236.189  mm,
	W =  90.000 deg,	P =   0.000 deg,	R =   90.000 deg
};
P[1320]{
   GP1:
	UF : 0, UT : 6,		CONFIG : 'N U T, 0, 0, 0',
	X =  342.831  mm,	Y =   -522.677  mm,	Z =   -235.930  mm,
	W =  90.000 deg,	P =   0.000 deg,	R =   90.000 deg
};
P[1321]{
   GP1:
	UF : 0, UT : 6,		CONFIG : 'N U T, 0, 0, 0',
	X =  343.741  mm,	Y =   -522.061  mm,	Z =   -236.148  mm,
	W =  90.000 deg,	P =   0.000 deg,	R =   90.000 deg
};
P[1322]{
   GP1:
	UF : 0, UT : 6,		CONFIG : 'N U T, 0, 0, 0',
	X =  347.154  mm,	Y =   -520.085  mm,	Z =   -236.164  mm,
	W =  90.000 deg,	P =   0.000 deg,	R =   90.000 deg
};
P[1323]{
   GP1:
	UF : 0, UT : 6,		CONFIG : 'N U T, 0, 0, 0',
	X =  349.167  mm,	Y =   -518.898  mm,	Z =   -236.221  mm,
	W =  90.000 deg,	P =   0.000 deg,	R =   90.000 deg
};
P[1324]{
   GP1:
	UF : 0, UT : 6,		CONFIG : 'N U T, 0, 0, 0',
	X =  352.757  mm,	Y =   -516.832  mm,	Z =   -236.203  mm,
	W =  90.000 deg,	P =   0.000 deg,	R =   90.000 deg
};
P[1325]{
   GP1:
	UF : 0, UT : 6,		CONFIG : 'N U T, 0, 0, 0',
	X =  356.030  mm,	Y =   -514.964  mm,	Z =   -236.152  mm,
	W =  90.000 deg,	P =   0.000 deg,	R =   90.000 deg
};
P[1326]{
   GP1:
	UF : 0, UT : 6,		CONFIG : 'N U T, 0, 0, 0',
	X =  357.181  mm,	Y =   -514.334  mm,	Z =   -236.069  mm,
	W =  90.000 deg,	P =   0.000 deg,	R =   90.000 deg
};
P[1327]{
   GP1:
	UF : 0, UT : 6,		CONFIG : 'N U T, 0, 0, 0',
	X =  358.019  mm,	Y =   -513.841  mm,	Z =   -236.091  mm,
	W =  90.000 deg,	P =   0.000 deg,	R =   90.000 deg
};
P[1328]{
   GP1:
	UF : 0, UT : 6,		CONFIG : 'N U T, 0, 0, 0',
	X =  358.836  mm,	Y =   -513.376  mm,	Z =   -236.075  mm,
	W =  90.000 deg,	P =   0.000 deg,	R =   90.000 deg
};
P[1329]{
   GP1:
	UF : 0, UT : 6,		CONFIG : 'N U T, 0, 0, 0',
	X =  359.384  mm,	Y =   -513.028  mm,	Z =   -236.152  mm,
	W =  90.000 deg,	P =   0.000 deg,	R =   90.000 deg
};
P[1330]{
   GP1:
	UF : 0, UT : 6,		CONFIG : 'N U T, 0, 0, 0',
	X =  360.335  mm,	Y =   -512.619  mm,	Z =   -235.811  mm,
	W =  90.000 deg,	P =   0.000 deg,	R =   90.000 deg
};
P[1331]{
   GP1:
	UF : 0, UT : 6,		CONFIG : 'N U T, 0, 0, 0',
	X =  362.804  mm,	Y =   -511.202  mm,	Z =   -235.789  mm,
	W =  90.000 deg,	P =   0.000 deg,	R =   90.000 deg
};
P[1332]{
   GP1:
	UF : 0, UT : 6,		CONFIG : 'N U T, 0, 0, 0',
	X =  364.805  mm,	Y =   -510.034  mm,	Z =   -235.820  mm,
	W =  90.000 deg,	P =   0.000 deg,	R =   90.000 deg
};
P[1333]{
   GP1:
	UF : 0, UT : 6,		CONFIG : 'N U T, 0, 0, 0',
	X =  365.931  mm,	Y =   -509.220  mm,	Z =   -236.218  mm,
	W =  90.000 deg,	P =   0.000 deg,	R =   90.000 deg
};
P[1334]{
   GP1:
	UF : 0, UT : 6,		CONFIG : 'N U T, 0, 0, 0',
	X =  366.787  mm,	Y =   -508.732  mm,	Z =   -236.203  mm,
	W =  90.000 deg,	P =   0.000 deg,	R =   90.000 deg
};
P[1335]{
   GP1:
	UF : 0, UT : 6,		CONFIG : 'N U T, 0, 0, 0',
	X =  369.185  mm,	Y =   -507.416  mm,	Z =   -236.037  mm,
	W =  90.000 deg,	P =   0.000 deg,	R =   90.000 deg
};
P[1336]{
   GP1:
	UF : 0, UT : 6,		CONFIG : 'N U T, 0, 0, 0',
	X =  370.161  mm,	Y =   -506.771  mm,	Z =   -236.235  mm,
	W =  90.000 deg,	P =   0.000 deg,	R =   90.000 deg
};
P[1337]{
   GP1:
	UF : 0, UT : 6,		CONFIG : 'N U T, 0, 0, 0',
	X =  370.741  mm,	Y =   -506.467  mm,	Z =   -236.161  mm,
	W =  90.000 deg,	P =   0.000 deg,	R =   90.000 deg
};
P[1338]{
   GP1:
	UF : 0, UT : 6,		CONFIG : 'N U T, 0, 0, 0',
	X =  373.216  mm,	Y =   -505.136  mm,	Z =   -235.923  mm,
	W =  90.000 deg,	P =   0.000 deg,	R =   90.000 deg
};
P[1339]{
   GP1:
	UF : 0, UT : 6,		CONFIG : 'N U T, 0, 0, 0',
	X =  373.769  mm,	Y =   -504.798  mm,	Z =   -235.968  mm,
	W =  90.000 deg,	P =   0.000 deg,	R =   90.000 deg
};
P[1340]{
   GP1:
	UF : 0, UT : 6,		CONFIG : 'N U T, 0, 0, 0',
	X =  375.268  mm,	Y =   -503.936  mm,	Z =   -235.961  mm,
	W =  90.000 deg,	P =   0.000 deg,	R =   90.000 deg
};
P[1341]{
   GP1:
	UF : 0, UT : 6,		CONFIG : 'N U T, 0, 0, 0',
	X =  376.365  mm,	Y =   -503.208  mm,	Z =   -236.189  mm,
	W =  90.000 deg,	P =   0.000 deg,	R =   90.000 deg
};
P[1342]{
   GP1:
	UF : 0, UT : 6,		CONFIG : 'N U T, 0, 0, 0',
	X =  377.812  mm,	Y =   -502.476  mm,	Z =   -235.937  mm,
	W =  90.000 deg,	P =   0.000 deg,	R =   90.000 deg
};
P[1343]{
   GP1:
	UF : 0, UT : 6,		CONFIG : 'N U T, 0, 0, 0',
	X =  378.644  mm,	Y =   -501.909  mm,	Z =   -236.149  mm,
	W =  90.000 deg,	P =   0.000 deg,	R =   90.000 deg
};
P[1344]{
   GP1:
	UF : 0, UT : 6,		CONFIG : 'N U T, 0, 0, 0',
	X =  382.006  mm,	Y =   -500.007  mm,	Z =   -236.051  mm,
	W =  90.000 deg,	P =   0.000 deg,	R =   90.000 deg
};
P[1345]{
   GP1:
	UF : 0, UT : 6,		CONFIG : 'N U T, 0, 0, 0',
	X =  384.094  mm,	Y =   -498.775  mm,	Z =   -236.118  mm,
	W =  90.000 deg,	P =   0.000 deg,	R =   90.000 deg
};
P[1346]{
   GP1:
	UF : 0, UT : 6,		CONFIG : 'N U T, 0, 0, 0',
	X =  385.040  mm,	Y =   -498.289  mm,	Z =   -235.969  mm,
	W =  90.000 deg,	P =   0.000 deg,	R =   90.000 deg
};
P[1347]{
   GP1:
	UF : 0, UT : 6,		CONFIG : 'N U T, 0, 0, 0',
	X =  387.969  mm,	Y =   -496.484  mm,	Z =   -236.245  mm,
	W =  90.000 deg,	P =   0.000 deg,	R =   90.000 deg
};
P[1348]{
   GP1:
	UF : 0, UT : 6,		CONFIG : 'N U T, 0, 0, 0',
	X =  388.653  mm,	Y =   -496.188  mm,	Z =   -236.005  mm,
	W =  90.000 deg,	P =   0.000 deg,	R =   90.000 deg
};
P[1349]{
   GP1:
	UF : 0, UT : 6,		CONFIG : 'N U T, 0, 0, 0',
	X =  389.771  mm,	Y =   -495.530  mm,	Z =   -236.036  mm,
	W =  90.000 deg,	P =   0.000 deg,	R =   90.000 deg
};
P[1350]{
   GP1:
	UF : 0, UT : 6,		CONFIG : 'N U T, 0, 0, 0',
	X =  391.734  mm,	Y =   -494.390  mm,	Z =   -236.054  mm,
	W =  90.000 deg,	P =   0.000 deg,	R =   90.000 deg
};
P[1351]{
   GP1:
	UF : 0, UT : 6,		CONFIG : 'N U T, 0, 0, 0',
	X =  393.563  mm,	Y =   -493.410  mm,	Z =   -235.867  mm,
	W =  90.000 deg,	P =   0.000 deg,	R =   90.000 deg
};
P[1352]{
   GP1:
	UF : 0, UT : 6,		CONFIG : 'N U T, 0, 0, 0',
	X =  395.191  mm,	Y =   -492.371  mm,	Z =   -236.108  mm,
	W =  90.000 deg,	P =   0.000 deg,	R =   90.000 deg
};
P[1353]{
   GP1:
	UF : 0, UT : 6,		CONFIG : 'N U T, 0, 0, 0',
	X =  395.783  mm,	Y =   -492.069  mm,	Z =   -236.013  mm,
	W =  90.000 deg,	P =   0.000 deg,	R =   90.000 deg
};
P[1354]{
   GP1:
	UF : 0, UT : 6,		CONFIG : 'N U T, 0, 0, 0',
	X =  396.375  mm,	Y =   -491.818  mm,	Z =   -235.791  mm,
	W =  90.000 deg,	P =   0.000 deg,	R =   90.000 deg
};
P[1355]{
   GP1:
	UF : 0, UT : 6,		CONFIG : 'N U T, 0, 0, 0',
	X =  397.057  mm,	Y =   -491.299  mm,	Z =   -236.097  mm,
	W =  90.000 deg,	P =   0.000 deg,	R =   90.000 deg
};
P[1356]{
   GP1:
	UF : 0, UT : 6,		CONFIG : 'N U T, 0, 0, 0',
	X =  398.898  mm,	Y =   -490.265  mm,	Z =   -236.024  mm,
	W =  90.000 deg,	P =   0.000 deg,	R =   90.000 deg
};
P[1357]{
   GP1:
	UF : 0, UT : 6,		CONFIG : 'N U T, 0, 0, 0',
	X =  399.925  mm,	Y =   -489.674  mm,	Z =   -236.019  mm,
	W =  90.000 deg,	P =   0.000 deg,	R =   90.000 deg
};
P[1358]{
   GP1:
	UF : 0, UT : 6,		CONFIG : 'N U T, 0, 0, 0',
	X =  401.212  mm,	Y =   -488.883  mm,	Z =   -236.137  mm,
	W =  90.000 deg,	P =   0.000 deg,	R =   90.000 deg
};
P[1359]{
   GP1:
	UF : 0, UT : 6,		CONFIG : 'N U T, 0, 0, 0',
	X =  403.329  mm,	Y =   -487.751  mm,	Z =   -235.916  mm,
	W =  90.000 deg,	P =   0.000 deg,	R =   90.000 deg
};
P[1360]{
   GP1:
	UF : 0, UT : 6,		CONFIG : 'N U T, 0, 0, 0',
	X =  403.952  mm,	Y =   -487.290  mm,	Z =   -236.163  mm,
	W =  90.000 deg,	P =   0.000 deg,	R =   90.000 deg
};
P[1361]{
   GP1:
	UF : 0, UT : 6,		CONFIG : 'N U T, 0, 0, 0',
	X =  404.904  mm,	Y =   -486.710  mm,	Z =   -236.237  mm,
	W =  90.000 deg,	P =   0.000 deg,	R =   90.000 deg
};
P[1362]{
   GP1:
	UF : 0, UT : 6,		CONFIG : 'N U T, 0, 0, 0',
	X =  406.898  mm,	Y =   -485.653  mm,	Z =   -236.006  mm,
	W =  90.000 deg,	P =   0.000 deg,	R =   90.000 deg
};
P[1363]{
   GP1:
	UF : 0, UT : 6,		CONFIG : 'N U T, 0, 0, 0',
	X =  407.911  mm,	Y =   -485.145  mm,	Z =   -235.822  mm,
	W =  90.000 deg,	P =   0.000 deg,	R =   90.000 deg
};
P[1364]{
   GP1:
	UF : 0, UT : 6,		CONFIG : 'N U T, 0, 0, 0',
	X =  408.697  mm,	Y =   -484.526  mm,	Z =   -236.222  mm,
	W =  90.000 deg,	P =   0.000 deg,	R =   90.000 deg
};
P[1365]{
   GP1:
	UF : 0, UT : 6,		CONFIG : 'N U T, 0, 0, 0',
	X =  409.952  mm,	Y =   -483.797  mm,	Z =   -236.231  mm,
	W =  90.000 deg,	P =   0.000 deg,	R =   90.000 deg
};
P[1366]{
   GP1:
	UF : 0, UT : 6,		CONFIG : 'N U T, 0, 0, 0',
	X =  411.074  mm,	Y =   -483.337  mm,	Z =   -235.777  mm,
	W =  90.000 deg,	P =   0.000 deg,	R =   90.000 deg
};
P[1367]{
   GP1:
	UF : 0, UT : 6,		CONFIG : 'N U T, 0, 0, 0',
	X =  412.204  mm,	Y =   -482.522  mm,	Z =   -236.171  mm,
	W =  90.000 deg,	P =   0.000 deg,	R =   90.000 deg
};
P[1368]{
   GP1:
	UF : 0, UT : 6,		CONFIG : 'N U T, 0, 0, 0',
	X =  413.895  mm,	Y =   -481.671  mm,	Z =   -235.868  mm,
	W =  90.000 deg,	P =   0.000 deg,	R =   90.000 deg
};
P[1369]{
   GP1:
	UF : 0, UT : 6,		CONFIG : 'N U T, 0, 0, 0',
	X =  415.738  mm,	Y =   -480.494  mm,	Z =   -236.139  mm,
	W =  90.000 deg,	P =   0.000 deg,	R =   90.000 deg
};
P[1370]{
   GP1:
	UF : 0, UT : 6,		CONFIG : 'N U T, 0, 0, 0',
	X =  416.784  mm,	Y =   -479.887  mm,	Z =   -236.148  mm,
	W =  90.000 deg,	P =   0.000 deg,	R =   90.000 deg
};
P[1371]{
   GP1:
	UF : 0, UT : 6,		CONFIG : 'N U T, 0, 0, 0',
	X =  419.161  mm,	Y =   -478.499  mm,	Z =   -236.184  mm,
	W =  90.000 deg,	P =   0.000 deg,	R =   90.000 deg
};
P[1372]{
   GP1:
	UF : 0, UT : 6,		CONFIG : 'N U T, 0, 0, 0',
	X =  420.459  mm,	Y =   -477.874  mm,	Z =   -235.882  mm,
	W =  90.000 deg,	P =   0.000 deg,	R =   90.000 deg
};
P[1373]{
   GP1:
	UF : 0, UT : 6,		CONFIG : 'N U T, 0, 0, 0',
	X =  422.127  mm,	Y =   -476.831  mm,	Z =   -236.078  mm,
	W =  90.000 deg,	P =   0.000 deg,	R =   90.000 deg
};
P[1374]{
   GP1:
	UF : 0, UT : 6,		CONFIG : 'N U T, 0, 0, 0',
	X =  423.415  mm,	Y =   -476.211  mm,	Z =   -235.778  mm,
	W =  90.000 deg,	P =   0.000 deg,	R =   90.000 deg
};
P[1375]{
   GP1:
	UF : 0, UT : 6,		CONFIG : 'N U T, 0, 0, 0',
	X =  424.988  mm,	Y =   -475.115  mm,	Z =   -236.232  mm,
	W =  90.000 deg,	P =   0.000 deg,	R =   90.000 deg
};
P[1376]{
   GP1:
	UF : 0, UT : 6,		CONFIG : 'N U T, 0, 0, 0',
	X =  426.209  mm,	Y =   -474.412  mm,	Z =   -236.229  mm,
	W =  90.000 deg,	P =   0.000 deg,	R =   90.000 deg
};
P[1377]{
   GP1:
	UF : 0, UT : 6,		CONFIG : 'N U T, 0, 0, 0',
	X =  426.886  mm,	Y =   -474.155  mm,	Z =   -235.903  mm,
	W =  90.000 deg,	P =   0.000 deg,	R =   90.000 deg
};
P[1378]{
   GP1:
	UF : 0, UT : 6,		CONFIG : 'N U T, 0, 0, 0',
	X =  427.565  mm,	Y =   -473.819  mm,	Z =   -235.766  mm,
	W =  90.000 deg,	P =   0.000 deg,	R =   90.000 deg
};
P[1379]{
   GP1:
	UF : 0, UT : 6,		CONFIG : 'N U T, 0, 0, 0',
	X =  428.364  mm,	Y =   -473.287  mm,	Z =   -235.939  mm,
	W =  90.000 deg,	P =   0.000 deg,	R =   90.000 deg
};
P[1380]{
   GP1:
	UF : 0, UT : 6,		CONFIG : 'N U T, 0, 0, 0',
	X =  430.727  mm,	Y =   -471.993  mm,	Z =   -235.767  mm,
	W =  90.000 deg,	P =   0.000 deg,	R =   90.000 deg
};
P[1381]{
   GP1:
	UF : 0, UT : 6,		CONFIG : 'N U T, 0, 0, 0',
	X =  433.236  mm,	Y =   -470.385  mm,	Z =   -236.155  mm,
	W =  90.000 deg,	P =   0.000 deg,	R =   90.000 deg
};
P[1382]{
   GP1:
	UF : 0, UT : 6,		CONFIG : 'N U T, 0, 0, 0',
	X =  434.178  mm,	Y =   -469.802  mm,	Z =   -236.249  mm,
	W =  90.000 deg,	P =   0.000 deg,	R =   90.000 deg
};
P[1383]{
   GP1:
	UF : 0, UT : 6,		CONFIG : 'N U T, 0, 0, 0',
	X =  439.088  mm,	Y =   -467.108  mm,	Z =   -235.908  mm,
	W =  90.000 deg,	P =   0.000 deg,	R =   90.000 deg
};
P[1384]{
   GP1:
	UF : 0, UT : 6,		CONFIG : 'N U T, 0, 0, 0',
	X =  442.078  mm,	Y =   -465.427  mm,	Z =   -235.796  mm,
	W =  90.000 deg,	P =   0.000 deg,	R =   90.000 deg
};
P[1385]{
   GP1:
	UF : 0, UT : 6,		CONFIG : 'N U T, 0, 0, 0',
	X =  442.626  mm,	Y =   -464.945  mm,	Z =   -236.199  mm,
	W =  90.000 deg,	P =   0.000 deg,	R =   90.000 deg
};
P[1386]{
   GP1:
	UF : 0, UT : 6,		CONFIG : 'N U T, 0, 0, 0',
	X =  445.138  mm,	Y =   -463.504  mm,	Z =   -236.176  mm,
	W =  90.000 deg,	P =   0.000 deg,	R =   90.000 deg
};
P[1387]{
   GP1:
	UF : 0, UT : 6,		CONFIG : 'N U T, 0, 0, 0',
	X =  446.827  mm,	Y =   -462.519  mm,	Z =   -236.199  mm,
	W =  90.000 deg,	P =   0.000 deg,	R =   90.000 deg
};
P[1388]{
   GP1:
	UF : 0, UT : 6,		CONFIG : 'N U T, 0, 0, 0',
	X =  448.090  mm,	Y =   -461.915  mm,	Z =   -235.896  mm,
	W =  90.000 deg,	P =   0.000 deg,	R =   90.000 deg
};
P[1389]{
   GP1:
	UF : 0, UT : 6,		CONFIG : 'N U T, 0, 0, 0',
	X =  450.063  mm,	Y =   -460.762  mm,	Z =   -235.929  mm,
	W =  90.000 deg,	P =   0.000 deg,	R =   90.000 deg
};
P[1390]{
   GP1:
	UF : 0, UT : 6,		CONFIG : 'N U T, 0, 0, 0',
	X =  454.885  mm,	Y =   -457.933  mm,	Z =   -236.037  mm,
	W =  90.000 deg,	P =   0.000 deg,	R =   90.000 deg
};
P[1391]{
   GP1:
	UF : 0, UT : 6,		CONFIG : 'N U T, 0, 0, 0',
	X =  455.876  mm,	Y =   -457.384  mm,	Z =   -235.981  mm,
	W =  90.000 deg,	P =   0.000 deg,	R =   90.000 deg
};
P[1392]{
   GP1:
	UF : 0, UT : 6,		CONFIG : 'N U T, 0, 0, 0',
	X =  457.280  mm,	Y =   -456.517  mm,	Z =   -236.120  mm,
	W =  90.000 deg,	P =   0.000 deg,	R =   90.000 deg
};
P[1393]{
   GP1:
	UF : 0, UT : 6,		CONFIG : 'N U T, 0, 0, 0',
	X =  458.154  mm,	Y =   -456.067  mm,	Z =   -235.987  mm,
	W =  90.000 deg,	P =   0.000 deg,	R =   90.000 deg
};
P[1394]{
   GP1:
	UF : 0, UT : 6,		CONFIG : 'N U T, 0, 0, 0',
	X =  458.736  mm,	Y =   -455.782  mm,	Z =   -235.861  mm,
	W =  90.000 deg,	P =   0.000 deg,	R =   90.000 deg
};
P[1395]{
   GP1:
	UF : 0, UT : 6,		CONFIG : 'N U T, 0, 0, 0',
	X =  459.445  mm,	Y =   -455.208  mm,	Z =   -236.262  mm,
	W =  90.000 deg,	P =   0.000 deg,	R =   90.000 deg
};
P[1396]{
   GP1:
	UF : 0, UT : 6,		CONFIG : 'N U T, 0, 0, 0',
	X =  462.501  mm,	Y =   -453.466  mm,	Z =   -236.208  mm,
	W =  90.000 deg,	P =   0.000 deg,	R =   90.000 deg
};
P[1397]{
   GP1:
	UF : 0, UT : 6,		CONFIG : 'N U T, 0, 0, 0',
	X =  464.409  mm,	Y =   -452.537  mm,	Z =   -235.787  mm,
	W =  90.000 deg,	P =   0.000 deg,	R =   90.000 deg
};
P[1398]{
   GP1:
	UF : 0, UT : 6,		CONFIG : 'N U T, 0, 0, 0',
	X =  466.034  mm,	Y =   -451.498  mm,	Z =   -236.031  mm,
	W =  90.000 deg,	P =   0.000 deg,	R =   90.000 deg
};
P[1399]{
   GP1:
	UF : 0, UT : 6,		CONFIG : 'N U T, 0, 0, 0',
	X =  469.539  mm,	Y =   -449.445  mm,	Z =   -236.103  mm,
	W =  90.000 deg,	P =   0.000 deg,	R =   90.000 deg
};
P[1400]{
   GP1:
	UF : 0, UT : 6,		CONFIG : 'N U T, 0, 0, 0',
	X =  471.370  mm,	Y =   -448.374  mm,	Z =   -236.138  mm,
	W =  90.000 deg,	P =   0.000 deg,	R =   90.000 deg
};
P[1401]{
   GP1:
	UF : 0, UT : 6,		CONFIG : 'N U T, 0, 0, 0',
	X =  473.342  mm,	Y =   -447.318  mm,	Z =   -235.937  mm,
	W =  90.000 deg,	P =   0.000 deg,	R =   90.000 deg
};
P[1402]{
   GP1:
	UF : 0, UT : 6,		CONFIG : 'N U T, 0, 0, 0',
	X =  475.559  mm,	Y =   -445.986  mm,	Z =   -236.063  mm,
	W =  90.000 deg,	P =   0.000 deg,	R =   90.000 deg
};
P[1403]{
   GP1:
	UF : 0, UT : 6,		CONFIG : 'N U T, 0, 0, 0',
	X =  477.475  mm,	Y =   -444.885  mm,	Z =   -236.051  mm,
	W =  90.000 deg,	P =   0.000 deg,	R =   90.000 deg
};
P[1404]{
   GP1:
	UF : 0, UT : 6,		CONFIG : 'N U T, 0, 0, 0',
	X =  480.365  mm,	Y =   -443.302  mm,	Z =   -235.842  mm,
	W =  90.000 deg,	P =   0.000 deg,	R =   90.000 deg
};
P[1405]{
   GP1:
	UF : 0, UT : 6,		CONFIG : 'N U T, 0, 0, 0',
	X =  480.787  mm,	Y =   -442.929  mm,	Z =   -236.155  mm,
	W =  90.000 deg,	P =   0.000 deg,	R =   90.000 deg
};
P[1406]{
   GP1:
	UF : 0, UT : 6,		CONFIG : 'N U T, 0, 0, 0',
	X =  481.795  mm,	Y =   -442.482  mm,	Z =   -235.830  mm,
	W =  90.000 deg,	P =   0.000 deg,	R =   90.000 deg
};
P[1407]{
   GP1:
	UF : 0, UT : 6,		CONFIG : 'N U T, 0, 0, 0',
	X =  482.369  mm,	Y =   -442.172  mm,	Z =   -235.775  mm,
	W =  90.000 deg,	P =   0.000 deg,	R =   90.000 deg
};
P[1408]{
   GP1:
	UF : 0, UT : 6,		CONFIG : 'N U T, 0, 0, 0',
	X =  483.508  mm,	Y =   -441.372  mm,	Z =   -236.122  mm,
	W =  90.000 deg,	P =   0.000 deg,	R =   90.000 deg
};
P[1409]{
   GP1:
	UF : 0, UT : 6,		CONFIG : 'N U T, 0, 0, 0',
	X =  484.395  mm,	Y =   -440.937  mm,	Z =   -235.933  mm,
	W =  90.000 deg,	P =   0.000 deg,	R =   90.000 deg
};
P[1410]{
   GP1:
	UF : 0, UT : 6,		CONFIG : 'N U T, 0, 0, 0',
	X =  493.607  mm,	Y =   -435.534  mm,	Z =   -236.136  mm,
	W =  90.000 deg,	P =   0.000 deg,	R =   90.000 deg
};
P[1411]{
   GP1:
	UF : 0, UT : 6,		CONFIG : 'N U T, 0, 0, 0',
	X =  494.690  mm,	Y =   -434.898  mm,	Z =   -236.165  mm,
	W =  90.000 deg,	P =   0.000 deg,	R =   90.000 deg
};
P[1412]{
   GP1:
	UF : 0, UT : 6,		CONFIG : 'N U T, 0, 0, 0',
	X =  495.486  mm,	Y =   -434.452  mm,	Z =   -236.133  mm,
	W =  90.000 deg,	P =   0.000 deg,	R =   90.000 deg
};
P[1413]{
   GP1:
	UF : 0, UT : 6,		CONFIG : 'N U T, 0, 0, 0',
	X =  501.371  mm,	Y =   -429.685  mm,	Z =   -236.260  mm,
	W =  90.000 deg,	P =   0.000 deg,	R =   90.000 deg
};
P[1414]{
   GP1:
	UF : 0, UT : 6,		CONFIG : 'N U T, 0, 0, 0',
	X =  502.086  mm,	Y =   -428.616  mm,	Z =   -236.164  mm,
	W =  90.000 deg,	P =   0.000 deg,	R =   90.000 deg
};
P[1415]{
   GP1:
	UF : 0, UT : 6,		CONFIG : 'N U T, 0, 0, 0',
	X =  503.490  mm,	Y =   -425.088  mm,	Z =   -236.147  mm,
	W =  90.000 deg,	P =   0.000 deg,	R =   90.000 deg
};
P[1416]{
   GP1:
	UF : 0, UT : 6,		CONFIG : 'N U T, 0, 0, 0',
	X =  503.787  mm,	Y =   -422.551  mm,	Z =   -236.120  mm,
	W =  90.000 deg,	P =   0.000 deg,	R =   90.000 deg
};
P[1417]{
   GP1:
	UF : 0, UT : 6,		CONFIG : 'N U T, 0, 0, 0',
	X =  503.943  mm,	Y =   -421.553  mm,	Z =   -235.775  mm,
	W =  90.000 deg,	P =   0.000 deg,	R =   90.000 deg
};
P[1418]{
   GP1:
	UF : 0, UT : 6,		CONFIG : 'N U T, 0, 0, 0',
	X =  503.776  mm,	Y =   -420.382  mm,	Z =   -235.795  mm,
	W =  90.000 deg,	P =   0.000 deg,	R =   90.000 deg
};
P[1419]{
   GP1:
	UF : 0, UT : 6,		CONFIG : 'N U T, 0, 0, 0',
	X =  502.567  mm,	Y =   -416.800  mm,	Z =   -235.937  mm,
	W =  90.000 deg,	P =   0.000 deg,	R =   90.000 deg
};
P[1420]{
   GP1:
	UF : 0, UT : 6,		CONFIG : 'N U T, 0, 0, 0',
	X =  502.027  mm,	Y =   -415.902  mm,	Z =   -236.236  mm,
	W =  90.000 deg,	P =   0.000 deg,	R =   90.000 deg
};
P[1421]{
   GP1:
	UF : 0, UT : 6,		CONFIG : 'N U T, 0, 0, 0',
	X =  501.509  mm,	Y =   -414.647  mm,	Z =   -235.780  mm,
	W =  90.000 deg,	P =   0.000 deg,	R =   90.000 deg
};
P[1422]{
   GP1:
	UF : 0, UT : 6,		CONFIG : 'N U T, 0, 0, 0',
	X =  500.751  mm,	Y =   -413.455  mm,	Z =   -235.950  mm,
	W =  90.000 deg,	P =   0.000 deg,	R =   90.000 deg
};
P[1423]{
   GP1:
	UF : 0, UT : 6,		CONFIG : 'N U T, 0, 0, 0',
	X =  500.064  mm,	Y =   -412.358  mm,	Z =   -236.082  mm,
	W =  90.000 deg,	P =   0.000 deg,	R =   90.000 deg
};
P[1424]{
   GP1:
	UF : 0, UT : 6,		CONFIG : 'N U T, 0, 0, 0',
	X =  498.507  mm,	Y =   -409.736  mm,	Z =   -236.184  mm,
	W =  90.000 deg,	P =   0.000 deg,	R =   90.000 deg
};
P[1425]{
   GP1:
	UF : 0, UT : 6,		CONFIG : 'N U T, 0, 0, 0',
	X =  498.135  mm,	Y =   -408.878  mm,	Z =   -235.884  mm,
	W =  90.000 deg,	P =   0.000 deg,	R =   90.000 deg
};
P[1426]{
   GP1:
	UF : 0, UT : 6,		CONFIG : 'N U T, 0, 0, 0',
	X =  496.210  mm,	Y =   -405.750  mm,	Z =   -236.173  mm,
	W =  90.000 deg,	P =   0.000 deg,	R =   90.000 deg
};
P[1427]{
   GP1:
	UF : 0, UT : 6,		CONFIG : 'N U T, 0, 0, 0',
	X =  494.639  mm,	Y =   -402.998  mm,	Z =   -236.133  mm,
	W =  90.000 deg,	P =   0.000 deg,	R =   90.000 deg
};
P[1428]{
   GP1:
	UF : 0, UT : 6,		CONFIG : 'N U T, 0, 0, 0',
	X =  491.870  mm,	Y =   -397.982  mm,	Z =   -235.821  mm,
	W =  90.000 deg,	P =   0.000 deg,	R =   90.000 deg
};
P[1429]{
   GP1:
	UF : 0, UT : 6,		CONFIG : 'N U T, 0, 0, 0',
	X =  491.287  mm,	Y =   -397.248  mm,	Z =   -236.208  mm,
	W =  90.000 deg,	P =   0.000 deg,	R =   90.000 deg
};
P[1430]{
   GP1:
	UF : 0, UT : 6,		CONFIG : 'N U T, 0, 0, 0',
	X =  490.763  mm,	Y =   -396.139  mm,	Z =   -235.927  mm,
	W =  90.000 deg,	P =   0.000 deg,	R =   90.000 deg
};
P[1431]{
   GP1:
	UF : 0, UT : 6,		CONFIG : 'N U T, 0, 0, 0',
	X =  489.685  mm,	Y =   -394.471  mm,	Z =   -236.207  mm,
	W =  90.000 deg,	P =   0.000 deg,	R =   90.000 deg
};
P[1432]{
   GP1:
	UF : 0, UT : 6,		CONFIG : 'N U T, 0, 0, 0',
	X =  489.004  mm,	Y =   -393.170  mm,	Z =   -236.035  mm,
	W =  90.000 deg,	P =   0.000 deg,	R =   90.000 deg
};
P[1433]{
   GP1:
	UF : 0, UT : 6,		CONFIG : 'N U T, 0, 0, 0',
	X =  487.863  mm,	Y =   -391.208  mm,	Z =   -236.054  mm,
	W =  90.000 deg,	P =   0.000 deg,	R =   90.000 deg
};
P[1434]{
   GP1:
	UF : 0, UT : 6,		CONFIG : 'N U T, 0, 0, 0',
	X =  486.334  mm,	Y =   -388.690  mm,	Z =   -236.237  mm,
	W =  90.000 deg,	P =   0.000 deg,	R =   90.000 deg
};
P[1435]{
   GP1:
	UF : 0, UT : 6,		CONFIG : 'N U T, 0, 0, 0',
	X =  485.304  mm,	Y =   -386.693  mm,	Z =   -235.939  mm,
	W =  90.000 deg,	P =   0.000 deg,	R =   90.000 deg
};
P[1436]{
   GP1:
	UF : 0, UT : 6,		CONFIG : 'N U T, 0, 0, 0',
	X =  484.893  mm,	Y =   -386.016  mm,	Z =   -235.984  mm,
	W =  90.000 deg,	P =   0.000 deg,	R =   90.000 deg
};
P[1437]{
   GP1:
	UF : 0, UT : 6,		CONFIG : 'N U T, 0, 0, 0',
	X =  484.497  mm,	Y =   -385.342  mm,	Z =   -236.003  mm,
	W =  90.000 deg,	P =   0.000 deg,	R =   90.000 deg
};
P[1438]{
   GP1:
	UF : 0, UT : 6,		CONFIG : 'N U T, 0, 0, 0',
	X =  483.642  mm,	Y =   -384.015  mm,	Z =   -236.218  mm,
	W =  90.000 deg,	P =   0.000 deg,	R =   90.000 deg
};
P[1439]{
   GP1:
	UF : 0, UT : 6,		CONFIG : 'N U T, 0, 0, 0',
	X =  483.324  mm,	Y =   -383.334  mm,	Z =   -236.037  mm,
	W =  90.000 deg,	P =   0.000 deg,	R =   90.000 deg
};
P[1440]{
   GP1:
	UF : 0, UT : 6,		CONFIG : 'N U T, 0, 0, 0',
	X =  482.982  mm,	Y =   -382.563  mm,	Z =   -235.786  mm,
	W =  90.000 deg,	P =   0.000 deg,	R =   90.000 deg
};
P[1441]{
   GP1:
	UF : 0, UT : 6,		CONFIG : 'N U T, 0, 0, 0',
	X =  482.333  mm,	Y =   -381.691  mm,	Z =   -236.140  mm,
	W =  90.000 deg,	P =   0.000 deg,	R =   90.000 deg
};
P[1442]{
   GP1:
	UF : 0, UT : 6,		CONFIG : 'N U T, 0, 0, 0',
	X =  481.019  mm,	Y =   -379.493  mm,	Z =   -236.251  mm,
	W =  90.000 deg,	P =   0.000 deg,	R =   90.000 deg
};
P[1443]{
   GP1:
	UF : 0, UT : 6,		CONFIG : 'N U T, 0, 0, 0',
	X =  479.633  mm,	Y =   -376.941  mm,	Z =   -236.036  mm,
	W =  90.000 deg,	P =   0.000 deg,	R =   90.000 deg
};
P[1444]{
   GP1:
	UF : 0, UT : 6,		CONFIG : 'N U T, 0, 0, 0',
	X =  479.309  mm,	Y =   -376.349  mm,	Z =   -235.992  mm,
	W =  90.000 deg,	P =   0.000 deg,	R =   90.000 deg
};
P[1445]{
   GP1:
	UF : 0, UT : 6,		CONFIG : 'N U T, 0, 0, 0',
	X =  478.404  mm,	Y =   -374.924  mm,	Z =   -236.192  mm,
	W =  90.000 deg,	P =   0.000 deg,	R =   90.000 deg
};
P[1446]{
   GP1:
	UF : 0, UT : 6,		CONFIG : 'N U T, 0, 0, 0',
	X =  476.232  mm,	Y =   -371.055  mm,	Z =   -236.043  mm,
	W =  90.000 deg,	P =   0.000 deg,	R =   90.000 deg
};
P[1447]{
   GP1:
	UF : 0, UT : 6,		CONFIG : 'N U T, 0, 0, 0',
	X =  474.537  mm,	Y =   -368.272  mm,	Z =   -236.256  mm,
	W =  90.000 deg,	P =   0.000 deg,	R =   90.000 deg
};
P[1448]{
   GP1:
	UF : 0, UT : 6,		CONFIG : 'N U T, 0, 0, 0',
	X =  472.913  mm,	Y =   -365.237  mm,	Z =   -235.945  mm,
	W =  90.000 deg,	P =   0.000 deg,	R =   90.000 deg
};
P[1449]{
   GP1:
	UF : 0, UT : 6,		CONFIG : 'N U T, 0, 0, 0',
	X =  472.386  mm,	Y =   -364.357  mm,	Z =   -235.991  mm,
	W =  90.000 deg,	P =   0.000 deg,	R =   90.000 deg
};
P[1450]{
   GP1:
	UF : 0, UT : 6,		CONFIG : 'N U T, 0, 0, 0',
	X =  471.989  mm,	Y =   -363.835  mm,	Z =   -236.221  mm,
	W =  90.000 deg,	P =   0.000 deg,	R =   90.000 deg
};
P[1451]{
   GP1:
	UF : 0, UT : 6,		CONFIG : 'N U T, 0, 0, 0',
	X =  471.449  mm,	Y =   -362.793  mm,	Z =   -236.073  mm,
	W =  90.000 deg,	P =   0.000 deg,	R =   90.000 deg
};
P[1452]{
   GP1:
	UF : 0, UT : 6,		CONFIG : 'N U T, 0, 0, 0',
	X =  470.745  mm,	Y =   -361.635  mm,	Z =   -236.161  mm,
	W =  90.000 deg,	P =   0.000 deg,	R =   90.000 deg
};
P[1453]{
   GP1:
	UF : 0, UT : 6,		CONFIG : 'N U T, 0, 0, 0',
	X =  469.696  mm,	Y =   -359.826  mm,	Z =   -236.171  mm,
	W =  90.000 deg,	P =   0.000 deg,	R =   90.000 deg
};
P[1454]{
   GP1:
	UF : 0, UT : 6,		CONFIG : 'N U T, 0, 0, 0',
	X =  468.767  mm,	Y =   -358.042  mm,	Z =   -235.924  mm,
	W =  90.000 deg,	P =   0.000 deg,	R =   90.000 deg
};
P[1455]{
   GP1:
	UF : 0, UT : 6,		CONFIG : 'N U T, 0, 0, 0',
	X =  467.703  mm,	Y =   -356.259  mm,	Z =   -236.006  mm,
	W =  90.000 deg,	P =   0.000 deg,	R =   90.000 deg
};
P[1456]{
   GP1:
	UF : 0, UT : 6,		CONFIG : 'N U T, 0, 0, 0',
	X =  466.876  mm,	Y =   -354.987  mm,	Z =   -236.231  mm,
	W =  90.000 deg,	P =   0.000 deg,	R =   90.000 deg
};
P[1457]{
   GP1:
	UF : 0, UT : 6,		CONFIG : 'N U T, 0, 0, 0',
	X =  466.291  mm,	Y =   -353.826  mm,	Z =   -236.026  mm,
	W =  90.000 deg,	P =   0.000 deg,	R =   90.000 deg
};
P[1458]{
   GP1:
	UF : 0, UT : 6,		CONFIG : 'N U T, 0, 0, 0',
	X =  465.009  mm,	Y =   -351.768  mm,	Z =   -236.252  mm,
	W =  90.000 deg,	P =   0.000 deg,	R =   90.000 deg
};
P[1459]{
   GP1:
	UF : 0, UT : 6,		CONFIG : 'N U T, 0, 0, 0',
	X =  464.591  mm,	Y =   -350.999  mm,	Z =   -236.191  mm,
	W =  90.000 deg,	P =   0.000 deg,	R =   90.000 deg
};
P[1460]{
   GP1:
	UF : 0, UT : 6,		CONFIG : 'N U T, 0, 0, 0',
	X =  463.595  mm,	Y =   -349.195  mm,	Z =   -236.079  mm,
	W =  90.000 deg,	P =   0.000 deg,	R =   90.000 deg
};
P[1461]{
   GP1:
	UF : 0, UT : 6,		CONFIG : 'N U T, 0, 0, 0',
	X =  463.089  mm,	Y =   -348.440  mm,	Z =   -236.248  mm,
	W =  90.000 deg,	P =   0.000 deg,	R =   90.000 deg
};
P[1462]{
   GP1:
	UF : 0, UT : 6,		CONFIG : 'N U T, 0, 0, 0',
	X =  462.640  mm,	Y =   -347.494  mm,	Z =   -236.014  mm,
	W =  90.000 deg,	P =   0.000 deg,	R =   90.000 deg
};
P[1463]{
   GP1:
	UF : 0, UT : 6,		CONFIG : 'N U T, 0, 0, 0',
	X =  461.755  mm,	Y =   -346.138  mm,	Z =   -236.261  mm,
	W =  90.000 deg,	P =   0.000 deg,	R =   90.000 deg
};
P[1464]{
   GP1:
	UF : 0, UT : 6,		CONFIG : 'N U T, 0, 0, 0',
	X =  460.704  mm,	Y =   -344.188  mm,	Z =   -236.079  mm,
	W =  90.000 deg,	P =   0.000 deg,	R =   90.000 deg
};
P[1465]{
   GP1:
	UF : 0, UT : 6,		CONFIG : 'N U T, 0, 0, 0',
	X =  459.501  mm,	Y =   -341.899  mm,	Z =   -235.791  mm,
	W =  90.000 deg,	P =   0.000 deg,	R =   90.000 deg
};
P[1466]{
   GP1:
	UF : 0, UT : 6,		CONFIG : 'N U T, 0, 0, 0',
	X =  458.900  mm,	Y =   -340.946  mm,	Z =   -235.915  mm,
	W =  90.000 deg,	P =   0.000 deg,	R =   90.000 deg
};
P[1467]{
   GP1:
	UF : 0, UT : 6,		CONFIG : 'N U T, 0, 0, 0',
	X =  458.293  mm,	Y =   -340.128  mm,	Z =   -236.243  mm,
	W =  90.000 deg,	P =   0.000 deg,	R =   90.000 deg
};
P[1468]{
   GP1:
	UF : 0, UT : 6,		CONFIG : 'N U T, 0, 0, 0',
	X =  457.137  mm,	Y =   -338.036  mm,	Z =   -236.113  mm,
	W =  90.000 deg,	P =   0.000 deg,	R =   90.000 deg
};
P[1469]{
   GP1:
	UF : 0, UT : 6,		CONFIG : 'N U T, 0, 0, 0',
	X =  456.482  mm,	Y =   -336.845  mm,	Z =   -236.037  mm,
	W =  90.000 deg,	P =   0.000 deg,	R =   90.000 deg
};
P[1470]{
   GP1:
	UF : 0, UT : 6,		CONFIG : 'N U T, 0, 0, 0',
	X =  456.051  mm,	Y =   -336.239  mm,	Z =   -236.233  mm,
	W =  90.000 deg,	P =   0.000 deg,	R =   90.000 deg
};
P[1471]{
   GP1:
	UF : 0, UT : 6,		CONFIG : 'N U T, 0, 0, 0',
	X =  454.647  mm,	Y =   -333.551  mm,	Z =   -235.872  mm,
	W =  90.000 deg,	P =   0.000 deg,	R =   90.000 deg
};
P[1472]{
   GP1:
	UF : 0, UT : 6,		CONFIG : 'N U T, 0, 0, 0',
	X =  454.146  mm,	Y =   -332.898  mm,	Z =   -236.173  mm,
	W =  90.000 deg,	P =   0.000 deg,	R =   90.000 deg
};
P[1473]{
   GP1:
	UF : 0, UT : 6,		CONFIG : 'N U T, 0, 0, 0',
	X =  453.247  mm,	Y =   -331.349  mm,	Z =   -236.186  mm,
	W =  90.000 deg,	P =   0.000 deg,	R =   90.000 deg
};
P[1474]{
   GP1:
	UF : 0, UT : 6,		CONFIG : 'N U T, 0, 0, 0',
	X =  453.051  mm,	Y =   -330.740  mm,	Z =   -235.808  mm,
	W =  90.000 deg,	P =   0.000 deg,	R =   90.000 deg
};
P[1475]{
   GP1:
	UF : 0, UT : 6,		CONFIG : 'N U T, 0, 0, 0',
	X =  451.791  mm,	Y =   -328.866  mm,	Z =   -236.239  mm,
	W =  90.000 deg,	P =   0.000 deg,	R =   90.000 deg
};
P[1476]{
   GP1:
	UF : 0, UT : 6,		CONFIG : 'N U T, 0, 0, 0',
	X =  451.415  mm,	Y =   -327.938  mm,	Z =   -235.851  mm,
	W =  90.000 deg,	P =   0.000 deg,	R =   90.000 deg
};
P[1477]{
   GP1:
	UF : 0, UT : 6,		CONFIG : 'N U T, 0, 0, 0',
	X =  450.389  mm,	Y =   -326.442  mm,	Z =   -236.246  mm,
	W =  90.000 deg,	P =   0.000 deg,	R =   90.000 deg
};
P[1478]{
   GP1:
	UF : 0, UT : 6,		CONFIG : 'N U T, 0, 0, 0',
	X =  450.072  mm,	Y =   -325.570  mm,	Z =   -235.794  mm,
	W =  90.000 deg,	P =   0.000 deg,	R =   90.000 deg
};
P[1479]{
   GP1:
	UF : 0, UT : 6,		CONFIG : 'N U T, 0, 0, 0',
	X =  448.973  mm,	Y =   -323.978  mm,	Z =   -236.228  mm,
	W =  90.000 deg,	P =   0.000 deg,	R =   90.000 deg
};
P[1480]{
   GP1:
	UF : 0, UT : 6,		CONFIG : 'N U T, 0, 0, 0',
	X =  447.200  mm,	Y =   -320.902  mm,	Z =   -236.222  mm,
	W =  90.000 deg,	P =   0.000 deg,	R =   90.000 deg
};
P[1481]{
   GP1:
	UF : 0, UT : 6,		CONFIG : 'N U T, 0, 0, 0',
	X =  445.841  mm,	Y =   -318.555  mm,	Z =   -236.231  mm,
	W =  90.000 deg,	P =   0.000 deg,	R =   90.000 deg
};
P[1482]{
   GP1:
	UF : 0, UT : 6,		CONFIG : 'N U T, 0, 0, 0',
	X =  445.418  mm,	Y =   -317.670  mm,	Z =   -236.017  mm,
	W =  90.000 deg,	P =   0.000 deg,	R =   90.000 deg
};
P[1483]{
   GP1:
	UF : 0, UT : 6,		CONFIG : 'N U T, 0, 0, 0',
	X =  444.001  mm,	Y =   -315.279  mm,	Z =   -236.105  mm,
	W =  90.000 deg,	P =   0.000 deg,	R =   90.000 deg
};
P[1484]{
   GP1:
	UF : 0, UT : 6,		CONFIG : 'N U T, 0, 0, 0',
	X =  442.340  mm,	Y =   -312.480  mm,	Z =   -236.214  mm,
	W =  90.000 deg,	P =   0.000 deg,	R =   90.000 deg
};
P[1485]{
   GP1:
	UF : 0, UT : 6,		CONFIG : 'N U T, 0, 0, 0',
	X =  440.973  mm,	Y =   -309.906  mm,	Z =   -235.927  mm,
	W =  90.000 deg,	P =   0.000 deg,	R =   90.000 deg
};
P[1486]{
   GP1:
	UF : 0, UT : 6,		CONFIG : 'N U T, 0, 0, 0',
	X =  440.412  mm,	Y =   -308.974  mm,	Z =   -235.981  mm,
	W =  90.000 deg,	P =   0.000 deg,	R =   90.000 deg
};
P[1487]{
   GP1:
	UF : 0, UT : 6,		CONFIG : 'N U T, 0, 0, 0',
	X =  439.918  mm,	Y =   -308.296  mm,	Z =   -236.229  mm,
	W =  90.000 deg,	P =   0.000 deg,	R =   90.000 deg
};
P[1488]{
   GP1:
	UF : 0, UT : 6,		CONFIG : 'N U T, 0, 0, 0',
	X =  437.104  mm,	Y =   -303.427  mm,	Z =   -236.235  mm,
	W =  90.000 deg,	P =   0.000 deg,	R =   90.000 deg
};
P[1489]{
   GP1:
	UF : 0, UT : 6,		CONFIG : 'N U T, 0, 0, 0',
	X =  436.579  mm,	Y =   -302.385  mm,	Z =   -236.050  mm,
	W =  90.000 deg,	P =   0.000 deg,	R =   90.000 deg
};
P[1490]{
   GP1:
	UF : 0, UT : 6,		CONFIG : 'N U T, 0, 0, 0',
	X =  435.638  mm,	Y =   -300.832  mm,	Z =   -236.157  mm,
	W =  90.000 deg,	P =   0.000 deg,	R =   90.000 deg
};
P[1491]{
   GP1:
	UF : 0, UT : 6,		CONFIG : 'N U T, 0, 0, 0',
	X =  435.193  mm,	Y =   -299.913  mm,	Z =   -235.950  mm,
	W =  90.000 deg,	P =   0.000 deg,	R =   90.000 deg
};
P[1492]{
   GP1:
	UF : 0, UT : 6,		CONFIG : 'N U T, 0, 0, 0',
	X =  434.306  mm,	Y =   -298.574  mm,	Z =   -236.225  mm,
	W =  90.000 deg,	P =   0.000 deg,	R =   90.000 deg
};
P[1493]{
   GP1:
	UF : 0, UT : 6,		CONFIG : 'N U T, 0, 0, 0',
	X =  433.514  mm,	Y =   -297.095  mm,	Z =   -236.075  mm,
	W =  90.000 deg,	P =   0.000 deg,	R =   90.000 deg
};
P[1494]{
   GP1:
	UF : 0, UT : 6,		CONFIG : 'N U T, 0, 0, 0',
	X =  432.995  mm,	Y =   -296.322  mm,	Z =   -236.252  mm,
	W =  90.000 deg,	P =   0.000 deg,	R =   90.000 deg
};
P[1495]{
   GP1:
	UF : 0, UT : 6,		CONFIG : 'N U T, 0, 0, 0',
	X =  432.605  mm,	Y =   -295.473  mm,	Z =   -236.008  mm,
	W =  90.000 deg,	P =   0.000 deg,	R =   90.000 deg
};
P[1496]{
   GP1:
	UF : 0, UT : 6,		CONFIG : 'N U T, 0, 0, 0',
	X =  430.299  mm,	Y =   -291.587  mm,	Z =   -236.161  mm,
	W =  90.000 deg,	P =   0.000 deg,	R =   90.000 deg
};
P[1497]{
   GP1:
	UF : 0, UT : 6,		CONFIG : 'N U T, 0, 0, 0',
	X =  429.850  mm,	Y =   -290.836  mm,	Z =   -236.197  mm,
	W =  90.000 deg,	P =   0.000 deg,	R =   90.000 deg
};
P[1498]{
   GP1:
	UF : 0, UT : 6,		CONFIG : 'N U T, 0, 0, 0',
	X =  428.081  mm,	Y =   -287.786  mm,	Z =   -236.217  mm,
	W =  90.000 deg,	P =   0.000 deg,	R =   90.000 deg
};
P[1499]{
   GP1:
	UF : 0, UT : 6,		CONFIG : 'N U T, 0, 0, 0',
	X =  426.184  mm,	Y =   -284.241  mm,	Z =   -235.855  mm,
	W =  90.000 deg,	P =   0.000 deg,	R =   90.000 deg
};
P[1500]{
   GP1:
	UF : 0, UT : 6,		CONFIG : 'N U T, 0, 0, 0',
	X =  424.899  mm,	Y =   -282.273  mm,	Z =   -236.213  mm,
	W =  90.000 deg,	P =   0.000 deg,	R =   90.000 deg
};
P[1501]{
   GP1:
	UF : 0, UT : 6,		CONFIG : 'N U T, 0, 0, 0',
	X =  422.960  mm,	Y =   -278.933  mm,	Z =   -236.239  mm,
	W =  90.000 deg,	P =   0.000 deg,	R =   90.000 deg
};
P[1502]{
   GP1:
	UF : 0, UT : 6,		CONFIG : 'N U T, 0, 0, 0',
	X =  421.968  mm,	Y =   -277.094  mm,	Z =   -236.069  mm,
	W =  90.000 deg,	P =   0.000 deg,	R =   90.000 deg
};
P[1503]{
   GP1:
	UF : 0, UT : 6,		CONFIG : 'N U T, 0, 0, 0',
	X =  420.506  mm,	Y =   -274.505  mm,	Z =   -235.991  mm,
	W =  90.000 deg,	P =   0.000 deg,	R =   90.000 deg
};
P[1504]{
   GP1:
	UF : 0, UT : 6,		CONFIG : 'N U T, 0, 0, 0',
	X =  418.260  mm,	Y =   -270.628  mm,	Z =   -236.010  mm,
	W =  90.000 deg,	P =   0.000 deg,	R =   90.000 deg
};
P[1505]{
   GP1:
	UF : 0, UT : 6,		CONFIG : 'N U T, 0, 0, 0',
	X =  417.918  mm,	Y =   -270.071  mm,	Z =   -236.057  mm,
	W =  90.000 deg,	P =   0.000 deg,	R =   90.000 deg
};
P[1506]{
   GP1:
	UF : 0, UT : 6,		CONFIG : 'N U T, 0, 0, 0',
	X =  416.905  mm,	Y =   -268.360  mm,	Z =   -236.120  mm,
	W =  90.000 deg,	P =   0.000 deg,	R =   90.000 deg
};
P[1507]{
   GP1:
	UF : 0, UT : 6,		CONFIG : 'N U T, 0, 0, 0',
	X =  415.790  mm,	Y =   -266.416  mm,	Z =   -236.101  mm,
	W =  90.000 deg,	P =   0.000 deg,	R =   90.000 deg
};
P[1508]{
   GP1:
	UF : 0, UT : 6,		CONFIG : 'N U T, 0, 0, 0',
	X =  412.830  mm,	Y =   -261.401  mm,	Z =   -236.257  mm,
	W =  90.000 deg,	P =   0.000 deg,	R =   90.000 deg
};
P[1509]{
   GP1:
	UF : 0, UT : 6,		CONFIG : 'N U T, 0, 0, 0',
	X =  412.227  mm,	Y =   -260.027  mm,	Z =   -235.795  mm,
	W =  90.000 deg,	P =   0.000 deg,	R =   90.000 deg
};
P[1510]{
   GP1:
	UF : 0, UT : 6,		CONFIG : 'N U T, 0, 0, 0',
	X =  409.230  mm,	Y =   -255.010  mm,	Z =   -236.040  mm,
	W =  90.000 deg,	P =   0.000 deg,	R =   90.000 deg
};
P[1511]{
   GP1:
	UF : 0, UT : 6,		CONFIG : 'N U T, 0, 0, 0',
	X =  408.186  mm,	Y =   -253.103  mm,	Z =   -235.901  mm,
	W =  90.000 deg,	P =   0.000 deg,	R =   90.000 deg
};
P[1512]{
   GP1:
	UF : 0, UT : 6,		CONFIG : 'N U T, 0, 0, 0',
	X =  406.843  mm,	Y =   -250.850  mm,	Z =   -236.001  mm,
	W =  90.000 deg,	P =   0.000 deg,	R =   90.000 deg
};
P[1513]{
   GP1:
	UF : 0, UT : 6,		CONFIG : 'N U T, 0, 0, 0',
	X =  403.954  mm,	Y =   -245.969  mm,	Z =   -236.175  mm,
	W =  90.000 deg,	P =   0.000 deg,	R =   90.000 deg
};
P[1514]{
   GP1:
	UF : 0, UT : 6,		CONFIG : 'N U T, 0, 0, 0',
	X =  403.237  mm,	Y =   -244.762  mm,	Z =   -236.224  mm,
	W =  90.000 deg,	P =   0.000 deg,	R =   90.000 deg
};
P[1515]{
   GP1:
	UF : 0, UT : 6,		CONFIG : 'N U T, 0, 0, 0',
	X =  402.871  mm,	Y =   -244.045  mm,	Z =   -236.107  mm,
	W =  90.000 deg,	P =   0.000 deg,	R =   90.000 deg
};
P[1516]{
   GP1:
	UF : 0, UT : 6,		CONFIG : 'N U T, 0, 0, 0',
	X =  401.992  mm,	Y =   -242.568  mm,	Z =   -236.169  mm,
	W =  90.000 deg,	P =   0.000 deg,	R =   90.000 deg
};
P[1517]{
   GP1:
	UF : 0, UT : 6,		CONFIG : 'N U T, 0, 0, 0',
	X =  401.454  mm,	Y =   -241.687  mm,	Z =   -236.241  mm,
	W =  90.000 deg,	P =   0.000 deg,	R =   90.000 deg
};
P[1518]{
   GP1:
	UF : 0, UT : 6,		CONFIG : 'N U T, 0, 0, 0',
	X =  401.098  mm,	Y =   -240.898  mm,	Z =   -235.999  mm,
	W =  90.000 deg,	P =   0.000 deg,	R =   90.000 deg
};
P[1519]{
   GP1:
	UF : 0, UT : 6,		CONFIG : 'N U T, 0, 0, 0',
	X =  400.564  mm,	Y =   -240.000  mm,	Z =   -236.036  mm,
	W =  90.000 deg,	P =   0.000 deg,	R =   90.000 deg
};
P[1520]{
   GP1:
	UF : 0, UT : 6,		CONFIG : 'N U T, 0, 0, 0',
	X =  399.685  mm,	Y =   -238.536  mm,	Z =   -236.120  mm,
	W =  90.000 deg,	P =   0.000 deg,	R =   90.000 deg
};
P[1521]{
   GP1:
	UF : 0, UT : 6,		CONFIG : 'N U T, 0, 0, 0',
	X =  398.765  mm,	Y =   -236.887  mm,	Z =   -236.042  mm,
	W =  90.000 deg,	P =   0.000 deg,	R =   90.000 deg
};
P[1522]{
   GP1:
	UF : 0, UT : 6,		CONFIG : 'N U T, 0, 0, 0',
	X =  398.278  mm,	Y =   -235.860  mm,	Z =   -235.784  mm,
	W =  90.000 deg,	P =   0.000 deg,	R =   90.000 deg
};
P[1523]{
   GP1:
	UF : 0, UT : 6,		CONFIG : 'N U T, 0, 0, 0',
	X =  396.435  mm,	Y =   -232.944  mm,	Z =   -236.170  mm,
	W =  90.000 deg,	P =   0.000 deg,	R =   90.000 deg
};
P[1524]{
   GP1:
	UF : 0, UT : 6,		CONFIG : 'N U T, 0, 0, 0',
	X =  395.504  mm,	Y =   -231.374  mm,	Z =   -236.229  mm,
	W =  90.000 deg,	P =   0.000 deg,	R =   90.000 deg
};
P[1525]{
   GP1:
	UF : 0, UT : 6,		CONFIG : 'N U T, 0, 0, 0',
	X =  395.074  mm,	Y =   -230.454  mm,	Z =   -235.985  mm,
	W =  90.000 deg,	P =   0.000 deg,	R =   90.000 deg
};
P[1526]{
   GP1:
	UF : 0, UT : 6,		CONFIG : 'N U T, 0, 0, 0',
	X =  394.275  mm,	Y =   -228.937  mm,	Z =   -235.797  mm,
	W =  90.000 deg,	P =   0.000 deg,	R =   90.000 deg
};
P[1527]{
   GP1:
	UF : 0, UT : 6,		CONFIG : 'N U T, 0, 0, 0',
	X =  393.835  mm,	Y =   -228.321  mm,	Z =   -236.002  mm,
	W =  90.000 deg,	P =   0.000 deg,	R =   90.000 deg
};
P[1528]{
   GP1:
	UF : 0, UT : 6,		CONFIG : 'N U T, 0, 0, 0',
	X =  393.146  mm,	Y =   -227.309  mm,	Z =   -236.255  mm,
	W =  90.000 deg,	P =   0.000 deg,	R =   90.000 deg
};
P[1529]{
   GP1:
	UF : 0, UT : 6,		CONFIG : 'N U T, 0, 0, 0',
	X =  392.427  mm,	Y =   -225.742  mm,	Z =   -235.806  mm,
	W =  90.000 deg,	P =   0.000 deg,	R =   90.000 deg
};
P[1530]{
   GP1:
	UF : 0, UT : 6,		CONFIG : 'N U T, 0, 0, 0',
	X =  389.578  mm,	Y =   -220.951  mm,	Z =   -236.007  mm,
	W =  90.000 deg,	P =   0.000 deg,	R =   90.000 deg
};
P[1531]{
   GP1:
	UF : 0, UT : 6,		CONFIG : 'N U T, 0, 0, 0',
	X =  389.058  mm,	Y =   -219.939  mm,	Z =   -235.851  mm,
	W =  90.000 deg,	P =   0.000 deg,	R =   90.000 deg
};
P[1532]{
   GP1:
	UF : 0, UT : 6,		CONFIG : 'N U T, 0, 0, 0',
	X =  387.191  mm,	Y =   -216.713  mm,	Z =   -235.860  mm,
	W =  90.000 deg,	P =   0.000 deg,	R =   90.000 deg
};
P[1533]{
   GP1:
	UF : 0, UT : 6,		CONFIG : 'N U T, 0, 0, 0',
	X =  383.632  mm,	Y =   -210.657  mm,	Z =   -236.010  mm,
	W =  90.000 deg,	P =   0.000 deg,	R =   90.000 deg
};
P[1534]{
   GP1:
	UF : 0, UT : 6,		CONFIG : 'N U T, 0, 0, 0',
	X =  383.089  mm,	Y =   -209.881  mm,	Z =   -236.241  mm,
	W =  90.000 deg,	P =   0.000 deg,	R =   90.000 deg
};
P[1535]{
   GP1:
	UF : 0, UT : 6,		CONFIG : 'N U T, 0, 0, 0',
	X =  382.024  mm,	Y =   -207.976  mm,	Z =   -236.157  mm,
	W =  90.000 deg,	P =   0.000 deg,	R =   90.000 deg
};
P[1536]{
   GP1:
	UF : 0, UT : 6,		CONFIG : 'N U T, 0, 0, 0',
	X =  380.879  mm,	Y =   -205.898  mm,	Z =   -236.024  mm,
	W =  90.000 deg,	P =   0.000 deg,	R =   90.000 deg
};
P[1537]{
   GP1:
	UF : 0, UT : 6,		CONFIG : 'N U T, 0, 0, 0',
	X =  379.546  mm,	Y =   -203.695  mm,	Z =   -236.174  mm,
	W =  90.000 deg,	P =   0.000 deg,	R =   90.000 deg
};
P[1538]{
   GP1:
	UF : 0, UT : 6,		CONFIG : 'N U T, 0, 0, 0',
	X =  378.877  mm,	Y =   -202.506  mm,	Z =   -236.128  mm,
	W =  90.000 deg,	P =   0.000 deg,	R =   90.000 deg
};
P[1539]{
   GP1:
	UF : 0, UT : 6,		CONFIG : 'N U T, 0, 0, 0',
	X =  377.434  mm,	Y =   -200.007  mm,	Z =   -236.130  mm,
	W =  90.000 deg,	P =   0.000 deg,	R =   90.000 deg
};
P[1540]{
   GP1:
	UF : 0, UT : 6,		CONFIG : 'N U T, 0, 0, 0',
	X =  377.085  mm,	Y =   -199.379  mm,	Z =   -236.095  mm,
	W =  90.000 deg,	P =   0.000 deg,	R =   90.000 deg
};
P[1541]{
   GP1:
	UF : 0, UT : 6,		CONFIG : 'N U T, 0, 0, 0',
	X =  375.858  mm,	Y =   -197.215  mm,	Z =   -236.043  mm,
	W =  90.000 deg,	P =   0.000 deg,	R =   90.000 deg
};
P[1542]{
   GP1:
	UF : 0, UT : 6,		CONFIG : 'N U T, 0, 0, 0',
	X =  371.444  mm,	Y =   -189.584  mm,	Z =   -236.064  mm,
	W =  90.000 deg,	P =   0.000 deg,	R =   90.000 deg
};
P[1543]{
   GP1:
	UF : 0, UT : 6,		CONFIG : 'N U T, 0, 0, 0',
	X =  370.368  mm,	Y =   -187.600  mm,	Z =   -235.892  mm,
	W =  90.000 deg,	P =   0.000 deg,	R =   90.000 deg
};
P[1544]{
   GP1:
	UF : 0, UT : 6,		CONFIG : 'N U T, 0, 0, 0',
	X =  368.994  mm,	Y =   -185.449  mm,	Z =   -236.214  mm,
	W =  90.000 deg,	P =   0.000 deg,	R =   90.000 deg
};
P[1545]{
   GP1:
	UF : 0, UT : 6,		CONFIG : 'N U T, 0, 0, 0',
	X =  367.915  mm,	Y =   -183.522  mm,	Z =   -236.133  mm,
	W =  90.000 deg,	P =   0.000 deg,	R =   90.000 deg
};
P[1546]{
   GP1:
	UF : 0, UT : 6,		CONFIG : 'N U T, 0, 0, 0',
	X =  367.612  mm,	Y =   -182.819  mm,	Z =   -235.883  mm,
	W =  90.000 deg,	P =   0.000 deg,	R =   90.000 deg
};
P[1547]{
   GP1:
	UF : 0, UT : 6,		CONFIG : 'N U T, 0, 0, 0',
	X =  364.111  mm,	Y =   -176.757  mm,	Z =   -235.886  mm,
	W =  90.000 deg,	P =   0.000 deg,	R =   90.000 deg
};
P[1548]{
   GP1:
	UF : 0, UT : 6,		CONFIG : 'N U T, 0, 0, 0',
	X =  361.125  mm,	Y =   -171.776  mm,	Z =   -236.149  mm,
	W =  90.000 deg,	P =   0.000 deg,	R =   90.000 deg
};
P[1549]{
   GP1:
	UF : 0, UT : 6,		CONFIG : 'N U T, 0, 0, 0',
	X =  358.906  mm,	Y =   -167.892  mm,	Z =   -236.094  mm,
	W =  90.000 deg,	P =   0.000 deg,	R =   90.000 deg
};
P[1550]{
   GP1:
	UF : 0, UT : 6,		CONFIG : 'N U T, 0, 0, 0',
	X =  356.038  mm,	Y =   -162.951  mm,	Z =   -236.129  mm,
	W =  90.000 deg,	P =   0.000 deg,	R =   90.000 deg
};
P[1551]{
   GP1:
	UF : 0, UT : 6,		CONFIG : 'N U T, 0, 0, 0',
	X =  354.732  mm,	Y =   -160.766  mm,	Z =   -236.239  mm,
	W =  90.000 deg,	P =   0.000 deg,	R =   90.000 deg
};
P[1552]{
   GP1:
	UF : 0, UT : 6,		CONFIG : 'N U T, 0, 0, 0',
	X =  353.869  mm,	Y =   -159.288  mm,	Z =   -236.260  mm,
	W =  90.000 deg,	P =   0.000 deg,	R =   90.000 deg
};
P[1553]{
   GP1:
	UF : 0, UT : 6,		CONFIG : 'N U T, 0, 0, 0',
	X =  350.471  mm,	Y =   -153.272  mm,	Z =   -236.078  mm,
	W =  90.000 deg,	P =   0.000 deg,	R =   90.000 deg
};
P[1554]{
   GP1:
	UF : 0, UT : 6,		CONFIG : 'N U T, 0, 0, 0',
	X =  349.723  mm,	Y =   -152.103  mm,	Z =   -236.255  mm,
	W =  90.000 deg,	P =   0.000 deg,	R =   90.000 deg
};
P[1555]{
   GP1:
	UF : 0, UT : 6,		CONFIG : 'N U T, 0, 0, 0',
	X =  348.267  mm,	Y =   -149.411  mm,	Z =   -236.017  mm,
	W =  90.000 deg,	P =   0.000 deg,	R =   90.000 deg
};
P[1556]{
   GP1:
	UF : 0, UT : 6,		CONFIG : 'N U T, 0, 0, 0',
	X =  347.032  mm,	Y =   -147.264  mm,	Z =   -236.007  mm,
	W =  90.000 deg,	P =   0.000 deg,	R =   90.000 deg
};
P[1557]{
   GP1:
	UF : 0, UT : 6,		CONFIG : 'N U T, 0, 0, 0',
	X =  344.262  mm,	Y =   -142.577  mm,	Z =   -236.161  mm,
	W =  90.000 deg,	P =   0.000 deg,	R =   90.000 deg
};
P[1558]{
   GP1:
	UF : 0, UT : 6,		CONFIG : 'N U T, 0, 0, 0',
	X =  343.139  mm,	Y =   -140.571  mm,	Z =   -235.898  mm,
	W =  90.000 deg,	P =   0.000 deg,	R =   90.000 deg
};
P[1559]{
   GP1:
	UF : 0, UT : 6,		CONFIG : 'N U T, 0, 0, 0',
	X =  342.580  mm,	Y =   -139.947  mm,	Z =   -236.127  mm,
	W =  90.000 deg,	P =   0.000 deg,	R =   90.000 deg
};
P[1560]{
   GP1:
	UF : 0, UT : 6,		CONFIG : 'N U T, 0, 0, 0',
	X =  342.085  mm,	Y =   -139.246  mm,	Z =   -236.094  mm,
	W =  90.000 deg,	P =   0.000 deg,	R =   90.000 deg
};
P[1561]{
   GP1:
	UF : 0, UT : 6,		CONFIG : 'N U T, 0, 0, 0',
	X =  341.506  mm,	Y =   -138.508  mm,	Z =   -235.946  mm,
	W =  90.000 deg,	P =   0.000 deg,	R =   90.000 deg
};
P[1562]{
   GP1:
	UF : 0, UT : 6,		CONFIG : 'N U T, 0, 0, 0',
	X =  340.743  mm,	Y =   -137.914  mm,	Z =   -236.128  mm,
	W =  90.000 deg,	P =   0.000 deg,	R =   90.000 deg
};
P[1563]{
   GP1:
	UF : 0, UT : 6,		CONFIG : 'N U T, 0, 0, 0',
	X =  339.447  mm,	Y =   -136.913  mm,	Z =   -236.218  mm,
	W =  90.000 deg,	P =   0.000 deg,	R =   90.000 deg
};
P[1564]{
   GP1:
	UF : 0, UT : 6,		CONFIG : 'N U T, 0, 0, 0',
	X =  338.577  mm,	Y =   -136.317  mm,	Z =   -236.085  mm,
	W =  90.000 deg,	P =   0.000 deg,	R =   90.000 deg
};
P[1565]{
   GP1:
	UF : 0, UT : 6,		CONFIG : 'N U T, 0, 0, 0',
	X =  335.791  mm,	Y =   -135.079  mm,	Z =   -235.939  mm,
	W =  90.000 deg,	P =   0.000 deg,	R =   90.000 deg
};
P[1566]{
   GP1:
	UF : 0, UT : 6,		CONFIG : 'N U T, 0, 0, 0',
	X =  334.841  mm,	Y =   -134.891  mm,	Z =   -236.057  mm,
	W =  90.000 deg,	P =   0.000 deg,	R =   90.000 deg
};
P[1567]{
   GP1:
	UF : 0, UT : 6,		CONFIG : 'N U T, 0, 0, 0',
	X =  333.673  mm,	Y =   -134.779  mm,	Z =   -236.169  mm,
	W =  90.000 deg,	P =   0.000 deg,	R =   90.000 deg
};
P[1568]{
   GP1:
	UF : 0, UT : 6,		CONFIG : 'N U T, 0, 0, 0',
	X =  331.872  mm,	Y =   -134.787  mm,	Z =   -236.252  mm,
	W =  90.000 deg,	P =   0.000 deg,	R =   90.000 deg
};
P[1569]{
   GP1:
	UF : 0, UT : 6,		CONFIG : 'N U T, 0, 0, 0',
	X =  330.732  mm,	Y =   -134.843  mm,	Z =   -236.144  mm,
	W =  90.000 deg,	P =   0.000 deg,	R =   90.000 deg
};
P[1570]{
   GP1:
	UF : 0, UT : 6,		CONFIG : 'N U T, 0, 0, 0',
	X =  330.113  mm,	Y =   -135.003  mm,	Z =   -236.220  mm,
	W =  90.000 deg,	P =   0.000 deg,	R =   90.000 deg
};
P[1571]{
   GP1:
	UF : 0, UT : 6,		CONFIG : 'N U T, 0, 0, 0',
	X =  327.814  mm,	Y =   -135.505  mm,	Z =   -235.881  mm,
	W =  90.000 deg,	P =   0.000 deg,	R =   90.000 deg
};
P[1572]{
   GP1:
	UF : 0, UT : 6,		CONFIG : 'N U T, 0, 0, 0',
	X =  326.279  mm,	Y =   -136.277  mm,	Z =   -236.071  mm,
	W =  90.000 deg,	P =   0.000 deg,	R =   90.000 deg
};
P[1573]{
   GP1:
	UF : 0, UT : 6,		CONFIG : 'N U T, 0, 0, 0',
	X =  320.577  mm,	Y =   -139.529  mm,	Z =   -236.099  mm,
	W =  90.000 deg,	P =   0.000 deg,	R =   90.000 deg
};
P[1574]{
   GP1:
	UF : 0, UT : 6,		CONFIG : 'N U T, 0, 0, 0',
	X =  318.856  mm,	Y =   -140.438  mm,	Z =   -235.891  mm,
	W =  90.000 deg,	P =   0.000 deg,	R =   90.000 deg
};
P[1575]{
   GP1:
	UF : 0, UT : 6,		CONFIG : 'N U T, 0, 0, 0',
	X =  318.009  mm,	Y =   -141.062  mm,	Z =   -236.220  mm,
	W =  90.000 deg,	P =   0.000 deg,	R =   90.000 deg
};
P[1576]{
   GP1:
	UF : 0, UT : 6,		CONFIG : 'N U T, 0, 0, 0',
	X =  317.193  mm,	Y =   -141.517  mm,	Z =   -236.179  mm,
	W =  90.000 deg,	P =   0.000 deg,	R =   90.000 deg
};
P[1577]{
   GP1:
	UF : 0, UT : 6,		CONFIG : 'N U T, 0, 0, 0',
	X =  314.066  mm,	Y =   -143.329  mm,	Z =   -236.196  mm,
	W =  90.000 deg,	P =   0.000 deg,	R =   90.000 deg
};
P[1578]{
   GP1:
	UF : 0, UT : 6,		CONFIG : 'N U T, 0, 0, 0',
	X =  313.250  mm,	Y =   -143.793  mm,	Z =   -236.178  mm,
	W =  90.000 deg,	P =   0.000 deg,	R =   90.000 deg
};
P[1579]{
   GP1:
	UF : 0, UT : 6,		CONFIG : 'N U T, 0, 0, 0',
	X =  312.553  mm,	Y =   -144.114  mm,	Z =   -235.981  mm,
	W =  90.000 deg,	P =   0.000 deg,	R =   90.000 deg
};
P[1580]{
   GP1:
	UF : 0, UT : 6,		CONFIG : 'N U T, 0, 0, 0',
	X =  311.510  mm,	Y =   -144.814  mm,	Z =   -236.218  mm,
	W =  90.000 deg,	P =   0.000 deg,	R =   90.000 deg
};
P[1581]{
   GP1:
	UF : 0, UT : 6,		CONFIG : 'N U T, 0, 0, 0',
	X =  308.829  mm,	Y =   -146.373  mm,	Z =   -236.244  mm,
	W =  90.000 deg,	P =   0.000 deg,	R =   90.000 deg
};
P[1582]{
   GP1:
	UF : 0, UT : 6,		CONFIG : 'N U T, 0, 0, 0',
	X =  305.966  mm,	Y =   -147.933  mm,	Z =   -236.020  mm,
	W =  90.000 deg,	P =   0.000 deg,	R =   90.000 deg
};
P[1583]{
   GP1:
	UF : 0, UT : 6,		CONFIG : 'N U T, 0, 0, 0',
	X =  304.183  mm,	Y =   -149.042  mm,	Z =   -236.210  mm,
	W =  90.000 deg,	P =   0.000 deg,	R =   90.000 deg
};
P[1584]{
   GP1:
	UF : 0, UT : 6,		CONFIG : 'N U T, 0, 0, 0',
	X =  297.401  mm,	Y =   -152.902  mm,	Z =   -236.079  mm,
	W =  90.000 deg,	P =   0.000 deg,	R =   90.000 deg
};
P[1585]{
   GP1:
	UF : 0, UT : 6,		CONFIG : 'N U T, 0, 0, 0',
	X =  296.221  mm,	Y =   -153.612  mm,	Z =   -236.148  mm,
	W =  90.000 deg,	P =   0.000 deg,	R =   90.000 deg
};
P[1586]{
   GP1:
	UF : 0, UT : 6,		CONFIG : 'N U T, 0, 0, 0',
	X =  295.539  mm,	Y =   -154.053  mm,	Z =   -236.259  mm,
	W =  90.000 deg,	P =   0.000 deg,	R =   90.000 deg
};
P[1587]{
   GP1:
	UF : 0, UT : 6,		CONFIG : 'N U T, 0, 0, 0',
	X =  293.360  mm,	Y =   -155.179  mm,	Z =   -235.938  mm,
	W =  90.000 deg,	P =   0.000 deg,	R =   90.000 deg
};
P[1588]{
   GP1:
	UF : 0, UT : 6,		CONFIG : 'N U T, 0, 0, 0',
	X =  290.547  mm,	Y =   -156.911  mm,	Z =   -236.202  mm,
	W =  90.000 deg,	P =   0.000 deg,	R =   90.000 deg
};
P[1589]{
   GP1:
	UF : 0, UT : 6,		CONFIG : 'N U T, 0, 0, 0',
	X =  288.220  mm,	Y =   -158.191  mm,	Z =   -236.046  mm,
	W =  90.000 deg,	P =   0.000 deg,	R =   90.000 deg
};
P[1590]{
   GP1:
	UF : 0, UT : 6,		CONFIG : 'N U T, 0, 0, 0',
	X =  285.132  mm,	Y =   -160.015  mm,	Z =   -236.148  mm,
	W =  90.000 deg,	P =   0.000 deg,	R =   90.000 deg
};
P[1591]{
   GP1:
	UF : 0, UT : 6,		CONFIG : 'N U T, 0, 0, 0',
	X =  283.394  mm,	Y =   -161.023  mm,	Z =   -236.157  mm,
	W =  90.000 deg,	P =   0.000 deg,	R =   90.000 deg
};
P[1592]{
   GP1:
	UF : 0, UT : 6,		CONFIG : 'N U T, 0, 0, 0',
	X =  277.986  mm,	Y =   -164.154  mm,	Z =   -236.180  mm,
	W =  90.000 deg,	P =   0.000 deg,	R =   90.000 deg
};
P[1593]{
   GP1:
	UF : 0, UT : 6,		CONFIG : 'N U T, 0, 0, 0',
	X =  275.580  mm,	Y =   -165.389  mm,	Z =   -235.805  mm,
	W =  90.000 deg,	P =   0.000 deg,	R =   90.000 deg
};
P[1594]{
   GP1:
	UF : 0, UT : 6,		CONFIG : 'N U T, 0, 0, 0',
	X =  274.939  mm,	Y =   -165.855  mm,	Z =   -236.037  mm,
	W =  90.000 deg,	P =   0.000 deg,	R =   90.000 deg
};
P[1595]{
   GP1:
	UF : 0, UT : 6,		CONFIG : 'N U T, 0, 0, 0',
	X =  273.899  mm,	Y =   -166.524  mm,	Z =   -236.202  mm,
	W =  90.000 deg,	P =   0.000 deg,	R =   90.000 deg
};
P[1596]{
   GP1:
	UF : 0, UT : 6,		CONFIG : 'N U T, 0, 0, 0',
	X =  273.201  mm,	Y =   -166.814  mm,	Z =   -235.930  mm,
	W =  90.000 deg,	P =   0.000 deg,	R =   90.000 deg
};
P[1597]{
   GP1:
	UF : 0, UT : 6,		CONFIG : 'N U T, 0, 0, 0',
	X =  270.621  mm,	Y =   -168.253  mm,	Z =   -235.806  mm,
	W =  90.000 deg,	P =   0.000 deg,	R =   90.000 deg
};
P[1598]{
   GP1:
	UF : 0, UT : 6,		CONFIG : 'N U T, 0, 0, 0',
	X =  269.332  mm,	Y =   -169.090  mm,	Z =   -236.033  mm,
	W =  90.000 deg,	P =   0.000 deg,	R =   90.000 deg
};
P[1599]{
   GP1:
	UF : 0, UT : 6,		CONFIG : 'N U T, 0, 0, 0',
	X =  268.290  mm,	Y =   -169.771  mm,	Z =   -236.223  mm,
	W =  90.000 deg,	P =   0.000 deg,	R =   90.000 deg
};
P[1600]{
   GP1:
	UF : 0, UT : 6,		CONFIG : 'N U T, 0, 0, 0',
	X =  267.307  mm,	Y =   -170.263  mm,	Z =   -236.040  mm,
	W =  90.000 deg,	P =   0.000 deg,	R =   90.000 deg
};
P[1601]{
   GP1:
	UF : 0, UT : 6,		CONFIG : 'N U T, 0, 0, 0',
	X =  264.439  mm,	Y =   -171.979  mm,	Z =   -236.185  mm,
	W =  90.000 deg,	P =   0.000 deg,	R =   90.000 deg
};
P[1602]{
   GP1:
	UF : 0, UT : 6,		CONFIG : 'N U T, 0, 0, 0',
	X =  263.829  mm,	Y =   -172.223  mm,	Z =   -235.924  mm,
	W =  90.000 deg,	P =   0.000 deg,	R =   90.000 deg
};
P[1603]{
   GP1:
	UF : 0, UT : 6,		CONFIG : 'N U T, 0, 0, 0',
	X =  262.750  mm,	Y =   -172.949  mm,	Z =   -236.173  mm,
	W =  90.000 deg,	P =   0.000 deg,	R =   90.000 deg
};
P[1604]{
   GP1:
	UF : 0, UT : 6,		CONFIG : 'N U T, 0, 0, 0',
	X =  257.108  mm,	Y =   -176.158  mm,	Z =   -236.056  mm,
	W =  90.000 deg,	P =   0.000 deg,	R =   90.000 deg
};
P[1605]{
   GP1:
	UF : 0, UT : 6,		CONFIG : 'N U T, 0, 0, 0',
	X =  255.758  mm,	Y =   -176.991  mm,	Z =   -236.186  mm,
	W =  90.000 deg,	P =   0.000 deg,	R =   90.000 deg
};
P[1606]{
   GP1:
	UF : 0, UT : 6,		CONFIG : 'N U T, 0, 0, 0',
	X =  255.088  mm,	Y =   -177.261  mm,	Z =   -235.902  mm,
	W =  90.000 deg,	P =   0.000 deg,	R =   90.000 deg
};
P[1607]{
   GP1:
	UF : 0, UT : 6,		CONFIG : 'N U T, 0, 0, 0',
	X =  254.014  mm,	Y =   -178.028  mm,	Z =   -236.258  mm,
	W =  90.000 deg,	P =   0.000 deg,	R =   90.000 deg
};
P[1608]{
   GP1:
	UF : 0, UT : 6,		CONFIG : 'N U T, 0, 0, 0',
	X =  251.531  mm,	Y =   -179.299  mm,	Z =   -235.862  mm,
	W =  90.000 deg,	P =   0.000 deg,	R =   90.000 deg
};
P[1609]{
   GP1:
	UF : 0, UT : 6,		CONFIG : 'N U T, 0, 0, 0',
	X =  250.849  mm,	Y =   -179.822  mm,	Z =   -236.178  mm,
	W =  90.000 deg,	P =   0.000 deg,	R =   90.000 deg
};
P[1610]{
   GP1:
	UF : 0, UT : 6,		CONFIG : 'N U T, 0, 0, 0',
	X =  248.064  mm,	Y =   -181.352  mm,	Z =   -235.984  mm,
	W =  90.000 deg,	P =   0.000 deg,	R =   90.000 deg
};
P[1611]{
   GP1:
	UF : 0, UT : 6,		CONFIG : 'N U T, 0, 0, 0',
	X =  247.392  mm,	Y =   -181.766  mm,	Z =   -236.049  mm,
	W =  90.000 deg,	P =   0.000 deg,	R =   90.000 deg
};
P[1612]{
   GP1:
	UF : 0, UT : 6,		CONFIG : 'N U T, 0, 0, 0',
	X =  244.453  mm,	Y =   -183.460  mm,	Z =   -236.045  mm,
	W =  90.000 deg,	P =   0.000 deg,	R =   90.000 deg
};
P[1613]{
   GP1:
	UF : 0, UT : 6,		CONFIG : 'N U T, 0, 0, 0',
	X =  238.622  mm,	Y =   -186.826  mm,	Z =   -236.043  mm,
	W =  90.000 deg,	P =   0.000 deg,	R =   90.000 deg
};
P[1614]{
   GP1:
	UF : 0, UT : 6,		CONFIG : 'N U T, 0, 0, 0',
	X =  237.753  mm,	Y =   -187.268  mm,	Z =   -235.896  mm,
	W =  90.000 deg,	P =   0.000 deg,	R =   90.000 deg
};
P[1615]{
   GP1:
	UF : 0, UT : 6,		CONFIG : 'N U T, 0, 0, 0',
	X =  237.145  mm,	Y =   -187.671  mm,	Z =   -236.022  mm,
	W =  90.000 deg,	P =   0.000 deg,	R =   90.000 deg
};
P[1616]{
   GP1:
	UF : 0, UT : 6,		CONFIG : 'N U T, 0, 0, 0',
	X =  232.443  mm,	Y =   -190.428  mm,	Z =   -236.124  mm,
	W =  90.000 deg,	P =   0.000 deg,	R =   90.000 deg
};
P[1617]{
   GP1:
	UF : 0, UT : 6,		CONFIG : 'N U T, 0, 0, 0',
	X =  231.517  mm,	Y =   -191.009  mm,	Z =   -236.238  mm,
	W =  90.000 deg,	P =   0.000 deg,	R =   90.000 deg
};
P[1618]{
   GP1:
	UF : 0, UT : 6,		CONFIG : 'N U T, 0, 0, 0',
	X =  230.852  mm,	Y =   -191.372  mm,	Z =   -236.187  mm,
	W =  90.000 deg,	P =   0.000 deg,	R =   90.000 deg
};
P[1619]{
   GP1:
	UF : 0, UT : 6,		CONFIG : 'N U T, 0, 0, 0',
	X =  230.182  mm,	Y =   -191.769  mm,	Z =   -236.210  mm,
	W =  90.000 deg,	P =   0.000 deg,	R =   90.000 deg
};
P[1620]{
   GP1:
	UF : 0, UT : 6,		CONFIG : 'N U T, 0, 0, 0',
	X =  226.559  mm,	Y =   -193.850  mm,	Z =   -236.186  mm,
	W =  90.000 deg,	P =   0.000 deg,	R =   90.000 deg
};
P[1621]{
   GP1:
	UF : 0, UT : 6,		CONFIG : 'N U T, 0, 0, 0',
	X =  225.729  mm,	Y =   -194.309  mm,	Z =   -236.135  mm,
	W =  90.000 deg,	P =   0.000 deg,	R =   90.000 deg
};
P[1622]{
   GP1:
	UF : 0, UT : 6,		CONFIG : 'N U T, 0, 0, 0',
	X =  223.917  mm,	Y =   -195.388  mm,	Z =   -236.215  mm,
	W =  90.000 deg,	P =   0.000 deg,	R =   90.000 deg
};
P[1623]{
   GP1:
	UF : 0, UT : 6,		CONFIG : 'N U T, 0, 0, 0',
	X =  222.484  mm,	Y =   -196.232  mm,	Z =   -236.254  mm,
	W =  90.000 deg,	P =   0.000 deg,	R =   90.000 deg
};
P[1624]{
   GP1:
	UF : 0, UT : 6,		CONFIG : 'N U T, 0, 0, 0',
	X =  221.399  mm,	Y =   -196.734  mm,	Z =   -235.953  mm,
	W =  90.000 deg,	P =   0.000 deg,	R =   90.000 deg
};
P[1625]{
   GP1:
	UF : 0, UT : 6,		CONFIG : 'N U T, 0, 0, 0',
	X =  220.565  mm,	Y =   -197.339  mm,	Z =   -236.253  mm,
	W =  90.000 deg,	P =   0.000 deg,	R =   90.000 deg
};
P[1626]{
   GP1:
	UF : 0, UT : 6,		CONFIG : 'N U T, 0, 0, 0',
	X =  219.701  mm,	Y =   -197.750  mm,	Z =   -236.038  mm,
	W =  90.000 deg,	P =   0.000 deg,	R =   90.000 deg
};
P[1627]{
   GP1:
	UF : 0, UT : 6,		CONFIG : 'N U T, 0, 0, 0',
	X =  218.470  mm,	Y =   -198.401  mm,	Z =   -235.896  mm,
	W =  90.000 deg,	P =   0.000 deg,	R =   90.000 deg
};
P[1628]{
   GP1:
	UF : 0, UT : 6,		CONFIG : 'N U T, 0, 0, 0',
	X =  217.609  mm,	Y =   -198.872  mm,	Z =   -235.831  mm,
	W =  90.000 deg,	P =   0.000 deg,	R =   90.000 deg
};
P[1629]{
   GP1:
	UF : 0, UT : 6,		CONFIG : 'N U T, 0, 0, 0',
	X =  215.081  mm,	Y =   -200.356  mm,	Z =   -235.891  mm,
	W =  90.000 deg,	P =   0.000 deg,	R =   90.000 deg
};
P[1630]{
   GP1:
	UF : 0, UT : 6,		CONFIG : 'N U T, 0, 0, 0',
	X =  212.664  mm,	Y =   -201.879  mm,	Z =   -236.200  mm,
	W =  90.000 deg,	P =   0.000 deg,	R =   90.000 deg
};
P[1631]{
   GP1:
	UF : 0, UT : 6,		CONFIG : 'N U T, 0, 0, 0',
	X =  210.426  mm,	Y =   -203.180  mm,	Z =   -236.221  mm,
	W =  90.000 deg,	P =   0.000 deg,	R =   90.000 deg
};
P[1632]{
   GP1:
	UF : 0, UT : 6,		CONFIG : 'N U T, 0, 0, 0',
	X =  209.402  mm,	Y =   -203.676  mm,	Z =   -235.990  mm,
	W =  90.000 deg,	P =   0.000 deg,	R =   90.000 deg
};
P[1633]{
   GP1:
	UF : 0, UT : 6,		CONFIG : 'N U T, 0, 0, 0',
	X =  207.230  mm,	Y =   -204.928  mm,	Z =   -235.987  mm,
	W =  90.000 deg,	P =   0.000 deg,	R =   90.000 deg
};
P[1634]{
   GP1:
	UF : 0, UT : 6,		CONFIG : 'N U T, 0, 0, 0',
	X =  206.599  mm,	Y =   -205.251  mm,	Z =   -235.885  mm,
	W =  90.000 deg,	P =   0.000 deg,	R =   90.000 deg
};
P[1635]{
   GP1:
	UF : 0, UT : 6,		CONFIG : 'N U T, 0, 0, 0',
	X =  205.983  mm,	Y =   -205.655  mm,	Z =   -236.001  mm,
	W =  90.000 deg,	P =   0.000 deg,	R =   90.000 deg
};
P[1636]{
   GP1:
	UF : 0, UT : 6,		CONFIG : 'N U T, 0, 0, 0',
	X =  203.848  mm,	Y =   -206.931  mm,	Z =   -236.105  mm,
	W =  90.000 deg,	P =   0.000 deg,	R =   90.000 deg
};
P[1637]{
   GP1:
	UF : 0, UT : 6,		CONFIG : 'N U T, 0, 0, 0',
	X =  202.883  mm,	Y =   -207.506  mm,	Z =   -236.150  mm,
	W =  90.000 deg,	P =   0.000 deg,	R =   90.000 deg
};
P[1638]{
   GP1:
	UF : 0, UT : 6,		CONFIG : 'N U T, 0, 0, 0',
	X =  201.148  mm,	Y =   -208.467  mm,	Z =   -236.049  mm,
	W =  90.000 deg,	P =   0.000 deg,	R =   90.000 deg
};
P[1639]{
   GP1:
	UF : 0, UT : 6,		CONFIG : 'N U T, 0, 0, 0',
	X =  199.810  mm,	Y =   -209.144  mm,	Z =   -235.818  mm,
	W =  90.000 deg,	P =   0.000 deg,	R =   90.000 deg
};
P[1640]{
   GP1:
	UF : 0, UT : 6,		CONFIG : 'N U T, 0, 0, 0',
	X =  198.203  mm,	Y =   -210.189  mm,	Z =   -236.102  mm,
	W =  90.000 deg,	P =   0.000 deg,	R =   90.000 deg
};
P[1641]{
   GP1:
	UF : 0, UT : 6,		CONFIG : 'N U T, 0, 0, 0',
	X =  197.583  mm,	Y =   -210.613  mm,	Z =   -236.263  mm,
	W =  90.000 deg,	P =   0.000 deg,	R =   90.000 deg
};
P[1642]{
   GP1:
	UF : 0, UT : 6,		CONFIG : 'N U T, 0, 0, 0',
	X =  195.751  mm,	Y =   -211.533  mm,	Z =   -235.929  mm,
	W =  90.000 deg,	P =   0.000 deg,	R =   90.000 deg
};
P[1643]{
   GP1:
	UF : 0, UT : 6,		CONFIG : 'N U T, 0, 0, 0',
	X =  194.806  mm,	Y =   -212.211  mm,	Z =   -236.250  mm,
	W =  90.000 deg,	P =   0.000 deg,	R =   90.000 deg
};
P[1644]{
   GP1:
	UF : 0, UT : 6,		CONFIG : 'N U T, 0, 0, 0',
	X =  193.660  mm,	Y =   -212.721  mm,	Z =   -235.883  mm,
	W =  90.000 deg,	P =   0.000 deg,	R =   90.000 deg
};
P[1645]{
   GP1:
	UF : 0, UT : 6,		CONFIG : 'N U T, 0, 0, 0',
	X =  191.475  mm,	Y =   -213.976  mm,	Z =   -235.864  mm,
	W =  90.000 deg,	P =   0.000 deg,	R =   90.000 deg
};
P[1646]{
   GP1:
	UF : 0, UT : 6,		CONFIG : 'N U T, 0, 0, 0',
	X =  190.496  mm,	Y =   -214.695  mm,	Z =   -236.240  mm,
	W =  90.000 deg,	P =   0.000 deg,	R =   90.000 deg
};
P[1647]{
   GP1:
	UF : 0, UT : 6,		CONFIG : 'N U T, 0, 0, 0',
	X =  189.353  mm,	Y =   -215.233  mm,	Z =   -235.942  mm,
	W =  90.000 deg,	P =   0.000 deg,	R =   90.000 deg
};
P[1648]{
   GP1:
	UF : 0, UT : 6,		CONFIG : 'N U T, 0, 0, 0',
	X =  187.581  mm,	Y =   -216.275  mm,	Z =   -235.989  mm,
	W =  90.000 deg,	P =   0.000 deg,	R =   90.000 deg
};
P[1649]{
   GP1:
	UF : 0, UT : 6,		CONFIG : 'N U T, 0, 0, 0',
	X =  186.678  mm,	Y =   -216.850  mm,	Z =   -236.119  mm,
	W =  90.000 deg,	P =   0.000 deg,	R =   90.000 deg
};
P[1650]{
   GP1:
	UF : 0, UT : 6,		CONFIG : 'N U T, 0, 0, 0',
	X =  185.648  mm,	Y =   -217.499  mm,	Z =   -236.251  mm,
	W =  90.000 deg,	P =   0.000 deg,	R =   90.000 deg
};
P[1651]{
   GP1:
	UF : 0, UT : 6,		CONFIG : 'N U T, 0, 0, 0',
	X =  183.841  mm,	Y =   -218.442  mm,	Z =   -236.010  mm,
	W =  90.000 deg,	P =   0.000 deg,	R =   90.000 deg
};
P[1652]{
   GP1:
	UF : 0, UT : 6,		CONFIG : 'N U T, 0, 0, 0',
	X =  182.443  mm,	Y =   -219.340  mm,	Z =   -236.228  mm,
	W =  90.000 deg,	P =   0.000 deg,	R =   90.000 deg
};
P[1653]{
   GP1:
	UF : 0, UT : 6,		CONFIG : 'N U T, 0, 0, 0',
	X =  179.934  mm,	Y =   -220.677  mm,	Z =   -235.957  mm,
	W =  90.000 deg,	P =   0.000 deg,	R =   90.000 deg
};
P[1654]{
   GP1:
	UF : 0, UT : 6,		CONFIG : 'N U T, 0, 0, 0',
	X =  177.647  mm,	Y =   -222.098  mm,	Z =   -236.202  mm,
	W =  90.000 deg,	P =   0.000 deg,	R =   90.000 deg
};
P[1655]{
   GP1:
	UF : 0, UT : 6,		CONFIG : 'N U T, 0, 0, 0',
	X =  175.862  mm,	Y =   -223.004  mm,	Z =   -235.897  mm,
	W =  90.000 deg,	P =   0.000 deg,	R =   90.000 deg
};
P[1656]{
   GP1:
	UF : 0, UT : 6,		CONFIG : 'N U T, 0, 0, 0',
	X =  175.057  mm,	Y =   -223.512  mm,	Z =   -236.004  mm,
	W =  90.000 deg,	P =   0.000 deg,	R =   90.000 deg
};
P[1657]{
   GP1:
	UF : 0, UT : 6,		CONFIG : 'N U T, 0, 0, 0',
	X =  170.716  mm,	Y =   -226.105  mm,	Z =   -236.214  mm,
	W =  90.000 deg,	P =   0.000 deg,	R =   90.000 deg
};
P[1658]{
   GP1:
	UF : 0, UT : 6,		CONFIG : 'N U T, 0, 0, 0',
	X =  168.211  mm,	Y =   -227.566  mm,	Z =   -236.248  mm,
	W =  90.000 deg,	P =   0.000 deg,	R =   90.000 deg
};
P[1659]{
   GP1:
	UF : 0, UT : 6,		CONFIG : 'N U T, 0, 0, 0',
	X =  167.336  mm,	Y =   -227.952  mm,	Z =   -235.959  mm,
	W =  90.000 deg,	P =   0.000 deg,	R =   90.000 deg
};
P[1660]{
   GP1:
	UF : 0, UT : 6,		CONFIG : 'N U T, 0, 0, 0',
	X =  165.023  mm,	Y =   -229.395  mm,	Z =   -236.220  mm,
	W =  90.000 deg,	P =   0.000 deg,	R =   90.000 deg
};
P[1661]{
   GP1:
	UF : 0, UT : 6,		CONFIG : 'N U T, 0, 0, 0',
	X =  164.294  mm,	Y =   -229.789  mm,	Z =   -236.153  mm,
	W =  90.000 deg,	P =   0.000 deg,	R =   90.000 deg
};
P[1662]{
   GP1:
	UF : 0, UT : 6,		CONFIG : 'N U T, 0, 0, 0',
	X =  163.660  mm,	Y =   -230.200  mm,	Z =   -236.263  mm,
	W =  90.000 deg,	P =   0.000 deg,	R =   90.000 deg
};
P[1663]{
   GP1:
	UF : 0, UT : 6,		CONFIG : 'N U T, 0, 0, 0',
	X =  161.734  mm,	Y =   -231.236  mm,	Z =   -236.080  mm,
	W =  90.000 deg,	P =   0.000 deg,	R =   90.000 deg
};
P[1664]{
   GP1:
	UF : 0, UT : 6,		CONFIG : 'N U T, 0, 0, 0',
	X =  160.385  mm,	Y =   -231.916  mm,	Z =   -235.838  mm,
	W =  90.000 deg,	P =   0.000 deg,	R =   90.000 deg
};
P[1665]{
   GP1:
	UF : 0, UT : 6,		CONFIG : 'N U T, 0, 0, 0',
	X =  155.746  mm,	Y =   -234.608  mm,	Z =   -235.873  mm,
	W =  90.000 deg,	P =   0.000 deg,	R =   90.000 deg
};
P[1666]{
   GP1:
	UF : 0, UT : 6,		CONFIG : 'N U T, 0, 0, 0',
	X =  154.862  mm,	Y =   -235.160  mm,	Z =   -235.974  mm,
	W =  90.000 deg,	P =   0.000 deg,	R =   90.000 deg
};
P[1667]{
   GP1:
	UF : 0, UT : 6,		CONFIG : 'N U T, 0, 0, 0',
	X =  153.080  mm,	Y =   -236.143  mm,	Z =   -235.861  mm,
	W =  90.000 deg,	P =   0.000 deg,	R =   90.000 deg
};
P[1668]{
   GP1:
	UF : 0, UT : 6,		CONFIG : 'N U T, 0, 0, 0',
	X =  151.825  mm,	Y =   -236.954  mm,	Z =   -236.070  mm,
	W =  90.000 deg,	P =   0.000 deg,	R =   90.000 deg
};
P[1669]{
   GP1:
	UF : 0, UT : 6,		CONFIG : 'N U T, 0, 0, 0',
	X =  150.266  mm,	Y =   -237.895  mm,	Z =   -236.170  mm,
	W =  90.000 deg,	P =   0.000 deg,	R =   90.000 deg
};
P[1670]{
   GP1:
	UF : 0, UT : 6,		CONFIG : 'N U T, 0, 0, 0',
	X =  148.626  mm,	Y =   -238.820  mm,	Z =   -236.117  mm,
	W =  90.000 deg,	P =   0.000 deg,	R =   90.000 deg
};
P[1671]{
   GP1:
	UF : 0, UT : 6,		CONFIG : 'N U T, 0, 0, 0',
	X =  148.088  mm,	Y =   -238.988  mm,	Z =   -235.770  mm,
	W =  90.000 deg,	P =   0.000 deg,	R =   90.000 deg
};
P[1672]{
   GP1:
	UF : 0, UT : 6,		CONFIG : 'N U T, 0, 0, 0',
	X =  145.272  mm,	Y =   -240.657  mm,	Z =   -235.874  mm,
	W =  90.000 deg,	P =   0.000 deg,	R =   90.000 deg
};
P[1673]{
   GP1:
	UF : 0, UT : 6,		CONFIG : 'N U T, 0, 0, 0',
	X =  144.713  mm,	Y =   -240.981  mm,	Z =   -235.879  mm,
	W =  90.000 deg,	P =   0.000 deg,	R =   90.000 deg
};
P[1674]{
   GP1:
	UF : 0, UT : 6,		CONFIG : 'N U T, 0, 0, 0',
	X =  142.594  mm,	Y =   -242.269  mm,	Z =   -236.034  mm,
	W =  90.000 deg,	P =   0.000 deg,	R =   90.000 deg
};
P[1675]{
   GP1:
	UF : 0, UT : 6,		CONFIG : 'N U T, 0, 0, 0',
	X =  141.204  mm,	Y =   -243.123  mm,	Z =   -236.160  mm,
	W =  90.000 deg,	P =   0.000 deg,	R =   90.000 deg
};
P[1676]{
   GP1:
	UF : 0, UT : 6,		CONFIG : 'N U T, 0, 0, 0',
	X =  134.413  mm,	Y =   -247.078  mm,	Z =   -236.241  mm,
	W =  90.000 deg,	P =   0.000 deg,	R =   90.000 deg
};
P[1677]{
   GP1:
	UF : 0, UT : 6,		CONFIG : 'N U T, 0, 0, 0',
	X =  133.189  mm,	Y =   -247.677  mm,	Z =   -235.980  mm,
	W =  90.000 deg,	P =   0.000 deg,	R =   90.000 deg
};
P[1678]{
   GP1:
	UF : 0, UT : 6,		CONFIG : 'N U T, 0, 0, 0',
	X =  132.385  mm,	Y =   -248.119  mm,	Z =   -235.927  mm,
	W =  90.000 deg,	P =   0.000 deg,	R =   90.000 deg
};
P[1679]{
   GP1:
	UF : 0, UT : 6,		CONFIG : 'N U T, 0, 0, 0',
	X =  131.644  mm,	Y =   -248.591  mm,	Z =   -236.035  mm,
	W =  90.000 deg,	P =   0.000 deg,	R =   90.000 deg
};
P[1680]{
   GP1:
	UF : 0, UT : 6,		CONFIG : 'N U T, 0, 0, 0',
	X =  130.373  mm,	Y =   -249.360  mm,	Z =   -236.121  mm,
	W =  90.000 deg,	P =   0.000 deg,	R =   90.000 deg
};
P[1681]{
   GP1:
	UF : 0, UT : 6,		CONFIG : 'N U T, 0, 0, 0',
	X =  126.528  mm,	Y =   -251.532  mm,	Z =   -236.003  mm,
	W =  90.000 deg,	P =   0.000 deg,	R =   90.000 deg
};
P[1682]{
   GP1:
	UF : 0, UT : 6,		CONFIG : 'N U T, 0, 0, 0',
	X =  124.220  mm,	Y =   -252.779  mm,	Z =   -235.795  mm,
	W =  90.000 deg,	P =   0.000 deg,	R =   90.000 deg
};
P[1683]{
   GP1:
	UF : 0, UT : 6,		CONFIG : 'N U T, 0, 0, 0',
	X =  118.465  mm,	Y =   -256.276  mm,	Z =   -236.219  mm,
	W =  90.000 deg,	P =   0.000 deg,	R =   90.000 deg
};
P[1684]{
   GP1:
	UF : 0, UT : 6,		CONFIG : 'N U T, 0, 0, 0',
	X =  117.055  mm,	Y =   -256.904  mm,	Z =   -235.765  mm,
	W =  90.000 deg,	P =   0.000 deg,	R =   90.000 deg
};
P[1685]{
   GP1:
	UF : 0, UT : 6,		CONFIG : 'N U T, 0, 0, 0',
	X =  116.477  mm,	Y =   -257.407  mm,	Z =   -236.175  mm,
	W =  90.000 deg,	P =   0.000 deg,	R =   90.000 deg
};
P[1686]{
   GP1:
	UF : 0, UT : 6,		CONFIG : 'N U T, 0, 0, 0',
	X =  114.900  mm,	Y =   -258.291  mm,	Z =   -236.112  mm,
	W =  90.000 deg,	P =   0.000 deg,	R =   90.000 deg
};
P[1687]{
   GP1:
	UF : 0, UT : 6,		CONFIG : 'N U T, 0, 0, 0',
	X =  114.102  mm,	Y =   -258.650  mm,	Z =   -235.865  mm,
	W =  90.000 deg,	P =   0.000 deg,	R =   90.000 deg
};
P[1688]{
   GP1:
	UF : 0, UT : 6,		CONFIG : 'N U T, 0, 0, 0',
	X =  111.110  mm,	Y =   -260.414  mm,	Z =   -235.952  mm,
	W =  90.000 deg,	P =   0.000 deg,	R =   90.000 deg
};
P[1689]{
   GP1:
	UF : 0, UT : 6,		CONFIG : 'N U T, 0, 0, 0',
	X =  110.514  mm,	Y =   -260.874  mm,	Z =   -236.236  mm,
	W =  90.000 deg,	P =   0.000 deg,	R =   90.000 deg
};
P[1690]{
   GP1:
	UF : 0, UT : 6,		CONFIG : 'N U T, 0, 0, 0',
	X =  109.604  mm,	Y =   -261.324  mm,	Z =   -236.052  mm,
	W =  90.000 deg,	P =   0.000 deg,	R =   90.000 deg
};
P[1691]{
   GP1:
	UF : 0, UT : 6,		CONFIG : 'N U T, 0, 0, 0',
	X =  107.200  mm,	Y =   -259.877  mm,	Z =   -229.170  mm,
	W =  90.000 deg,	P =   0.000 deg,	R =   90.000 deg
};
P[1692]{
   GP1:
	UF : 0, UT : 6,		CONFIG : 'N U T, 0, 0, 0',
	X =  106.066  mm,	Y =   -260.533  mm,	Z =   -229.172  mm,
	W =  90.000 deg,	P =   0.000 deg,	R =   90.000 deg
};
P[1693]{
   GP1:
	UF : 0, UT : 6,		CONFIG : 'N U T, 0, 0, 0',
	X =  104.641  mm,	Y =   -261.418  mm,	Z =   -229.323  mm,
	W =  90.000 deg,	P =   0.000 deg,	R =   90.000 deg
};
P[1694]{
   GP1:
	UF : 0, UT : 6,		CONFIG : 'N U T, 0, 0, 0',
	X =  103.260  mm,	Y =   -262.135  mm,	Z =   -229.128  mm,
	W =  90.000 deg,	P =   0.000 deg,	R =   90.000 deg
};
P[1695]{
   GP1:
	UF : 0, UT : 6,		CONFIG : 'N U T, 0, 0, 0',
	X =  101.827  mm,	Y =   -262.999  mm,	Z =   -229.218  mm,
	W =  90.000 deg,	P =   0.000 deg,	R =   90.000 deg
};
P[1696]{
   GP1:
	UF : 0, UT : 6,		CONFIG : 'N U T, 0, 0, 0',
	X =  100.336  mm,	Y =   -263.866  mm,	Z =   -229.231  mm,
	W =  90.000 deg,	P =   0.000 deg,	R =   90.000 deg
};
P[1697]{
   GP1:
	UF : 0, UT : 6,		CONFIG : 'N U T, 0, 0, 0',
	X =  99.594  mm,	Y =   -264.258  mm,	Z =   -229.143  mm,
	W =  90.000 deg,	P =   0.000 deg,	R =   90.000 deg
};
P[1698]{
   GP1:
	UF : 0, UT : 6,		CONFIG : 'N U T, 0, 0, 0',
	X =  98.829  mm,	Y =   -264.730  mm,	Z =   -229.218  mm,
	W =  90.000 deg,	P =   0.000 deg,	R =   90.000 deg
};
P[1699]{
   GP1:
	UF : 0, UT : 6,		CONFIG : 'N U T, 0, 0, 0',
	X =  96.716  mm,	Y =   -265.843  mm,	Z =   -228.958  mm,
	W =  90.000 deg,	P =   0.000 deg,	R =   90.000 deg
};
P[1700]{
   GP1:
	UF : 0, UT : 6,		CONFIG : 'N U T, 0, 0, 0',
	X =  95.303  mm,	Y =   -266.797  mm,	Z =   -229.294  mm,
	W =  90.000 deg,	P =   0.000 deg,	R =   90.000 deg
};
P[1701]{
   GP1:
	UF : 0, UT : 6,		CONFIG : 'N U T, 0, 0, 0',
	X =  93.990  mm,	Y =   -267.396  mm,	Z =   -228.909  mm,
	W =  90.000 deg,	P =   0.000 deg,	R =   90.000 deg
};
P[1702]{
   GP1:
	UF : 0, UT : 6,		CONFIG : 'N U T, 0, 0, 0',
	X =  91.593  mm,	Y =   -268.821  mm,	Z =   -229.009  mm,
	W =  90.000 deg,	P =   0.000 deg,	R =   90.000 deg
};
P[1703]{
   GP1:
	UF : 0, UT : 6,		CONFIG : 'N U T, 0, 0, 0',
	X =  91.045  mm,	Y =   -269.247  mm,	Z =   -229.272  mm,
	W =  90.000 deg,	P =   0.000 deg,	R =   90.000 deg
};
P[1704]{
   GP1:
	UF : 0, UT : 6,		CONFIG : 'N U T, 0, 0, 0',
	X =  90.331  mm,	Y =   -269.506  mm,	Z =   -228.899  mm,
	W =  90.000 deg,	P =   0.000 deg,	R =   90.000 deg
};
P[1705]{
   GP1:
	UF : 0, UT : 6,		CONFIG : 'N U T, 0, 0, 0',
	X =  88.025  mm,	Y =   -270.934  mm,	Z =   -229.135  mm,
	W =  90.000 deg,	P =   0.000 deg,	R =   90.000 deg
};
P[1706]{
   GP1:
	UF : 0, UT : 6,		CONFIG : 'N U T, 0, 0, 0',
	X =  87.040  mm,	Y =   -271.443  mm,	Z =   -228.990  mm,
	W =  90.000 deg,	P =   0.000 deg,	R =   90.000 deg
};
P[1707]{
   GP1:
	UF : 0, UT : 6,		CONFIG : 'N U T, 0, 0, 0',
	X =  85.101  mm,	Y =   -272.713  mm,	Z =   -229.356  mm,
	W =  90.000 deg,	P =   0.000 deg,	R =   90.000 deg
};
P[1708]{
   GP1:
	UF : 0, UT : 6,		CONFIG : 'N U T, 0, 0, 0',
	X =  82.612  mm,	Y =   -274.101  mm,	Z =   -229.237  mm,
	W =  90.000 deg,	P =   0.000 deg,	R =   90.000 deg
};
P[1709]{
   GP1:
	UF : 0, UT : 6,		CONFIG : 'N U T, 0, 0, 0',
	X =  81.482  mm,	Y =   -274.692  mm,	Z =   -229.088  mm,
	W =  90.000 deg,	P =   0.000 deg,	R =   90.000 deg
};
P[1710]{
   GP1:
	UF : 0, UT : 6,		CONFIG : 'N U T, 0, 0, 0',
	X =  79.166  mm,	Y =   -275.986  mm,	Z =   -228.982  mm,
	W =  90.000 deg,	P =   0.000 deg,	R =   90.000 deg
};
P[1711]{
   GP1:
	UF : 0, UT : 6,		CONFIG : 'N U T, 0, 0, 0',
	X =  77.547  mm,	Y =   -277.016  mm,	Z =   -229.213  mm,
	W =  90.000 deg,	P =   0.000 deg,	R =   90.000 deg
};
P[1712]{
   GP1:
	UF : 0, UT : 6,		CONFIG : 'N U T, 0, 0, 0',
	X =  75.851  mm,	Y =   -277.984  mm,	Z =   -229.188  mm,
	W =  90.000 deg,	P =   0.000 deg,	R =   90.000 deg
};
P[1713]{
   GP1:
	UF : 0, UT : 6,		CONFIG : 'N U T, 0, 0, 0',
	X =  73.182  mm,	Y =   -279.507  mm,	Z =   -229.142  mm,
	W =  90.000 deg,	P =   0.000 deg,	R =   90.000 deg
};
P[1714]{
   GP1:
	UF : 0, UT : 6,		CONFIG : 'N U T, 0, 0, 0',
	X =  71.099  mm,	Y =   -280.688  mm,	Z =   -229.089  mm,
	W =  90.000 deg,	P =   0.000 deg,	R =   90.000 deg
};
P[1715]{
   GP1:
	UF : 0, UT : 6,		CONFIG : 'N U T, 0, 0, 0',
	X =  69.665  mm,	Y =   -281.581  mm,	Z =   -229.246  mm,
	W =  90.000 deg,	P =   0.000 deg,	R =   90.000 deg
};
P[1716]{
   GP1:
	UF : 0, UT : 6,		CONFIG : 'N U T, 0, 0, 0',
	X =  68.447  mm,	Y =   -282.158  mm,	Z =   -228.943  mm,
	W =  90.000 deg,	P =   0.000 deg,	R =   90.000 deg
};
P[1717]{
   GP1:
	UF : 0, UT : 6,		CONFIG : 'N U T, 0, 0, 0',
	X =  67.511  mm,	Y =   -282.852  mm,	Z =   -229.314  mm,
